LIN {X 0,Y 353.225,Z 325.982,A -85,B 0,C 180,E1 -13406.578,E2 -13406.578} C_VEL
LIN {X 0,Y 353.193,Z 327.589,A -85,B 0,C 180,E1 -13408.86,E2 -13408.86} C_VEL
LIN {X 0,Y 353.218,Z 327.806,A -85,B 0,C 180,E1 -13410,E2 -13410} C_VEL
LIN {X 0,Y 353.193,Z 327.588,A -85,B 0,C 180,E1 -13411.14,E2 -13411.14} C_VEL
LIN {X 0,Y 353.225,Z 325.981,A -85,B 0,C 180,E1 -13413.422,E2 -13413.422} C_VEL
LIN {X 0,Y 353.299,Z 324.582,A -85,B 0,C 180,E1 -13414.564,E2 -13414.564} C_VEL
LIN {X 0,Y 353.388,Z 322.015,A -85,B 0,C 180,E1 -13416.079,E2 -13416.079} C_VEL
LIN {X 0,Y 353.694,Z 317.659,A -85,B 0,C 180,E1 -13417.995,E2 -13417.995} C_VEL
LIN {X 0,Y 354.272,Z 311.542,A -85,B 0,C 180,E1 -13419.996,E2 -13419.996} C_VEL
LIN {X 0,Y 354.955,Z 304.859,A -85,B 0,C 180,E1 -13421.709,E2 -13421.709} C_VEL
LIN {X 0,Y 355.96,Z 296.573,A -85,B 0,C 180,E1 -13423.414,E2 -13423.414} C_VEL
LIN {X 0,Y 356.926,Z 288.08,A -85,B 0,C 180,E1 -13424.831,E2 -13424.831} C_VEL
LIN {X 0,Y 357.965,Z 277.583,A -85,B 0,C 180,E1 -13426.246,E2 -13426.246} C_VEL
LIN {X 0,Y 359.229,Z 265.776,A -85,B 0,C 180,E1 -13427.505,E2 -13427.505} C_VEL
LIN {X 0,Y 359.965,Z 256.498,A -85,B 0,C 180,E1 -13428.294,E2 -13428.294} C_VEL
LIN {X 0,Y 358.531,Z 244.559,A -85,B 0,C 180,E1 -13429.213,E2 -13429.213} C_VEL
LIN {X 0,Y 356.413,Z 231.564,A -85,B 0,C 180,E1 -13429.992,E2 -13429.992} C_VEL
LIN {X 0,Y 354.223,Z 221.02,A -85,B 0,C 180,E1 -13430.496,E2 -13430.496} C_VEL
LIN {X 0,Y 354.747,Z 213.839,A -85,B 0,C 180,E1 -13434.584,E2 -13434.584} C_VEL
LIN {X 0,Y 355.283,Z 207.313,A -85,B 0,C 180,E1 -13438.343,E2 -13438.343} C_VEL
LIN {X 0,Y 355.9,Z 201.27,A -85,B 0,C 180,E1 -13441.883,E2 -13441.883} C_VEL
LIN {X 0,Y 356.363,Z 196.323,A -85,B 0,C 180,E1 -13444.884,E2 -13444.884} C_VEL
LIN {X 0,Y 356.215,Z 191.647,A -85,B 0,C 180,E1 -13447.89,E2 -13447.89} C_VEL
LIN {X 0,Y 355.436,Z 186.73,A -85,B 0,C 180,E1 -13451.291,E2 -13451.291} C_VEL
LIN {X 0,Y 354.794,Z 183.295,A -85,B 0,C 180,E1 -13453.892,E2 -13453.892} C_VEL
LIN {X 0,Y 354.793,Z 183.288,A -85,B 0,C 180,E1 -13457.662,E2 -13457.662} C_VEL
LIN {X 0,Y 354.783,Z 183.293,A -85,B 0,C 180,E1 -13460.662,E2 -13460.662} C_VEL
LIN {X 0,Y 354.819,Z 183.29,A -85,B 0,C 180,E1 -13464.301,E2 -13464.301} C_VEL
LIN {X 0,Y 354.785,Z 183.29,A -85,B 0,C 180,E1 -13467.666,E2 -13467.666} C_VEL
LIN {X 0,Y 354.844,Z 183.283,A -85,B 0,C 180,E1 -13471.618,E2 -13471.618} C_VEL
LIN {X 0,Y 354.896,Z 183.278,A -85,B 0,C 180,E1 -13474.172,E2 -13474.172} C_VEL
LIN {X 0,Y 354.813,Z 183.29,A -85,B 0,C 180,E1 -13477.893,E2 -13477.893} C_VEL
LIN {X 0,Y 354.921,Z 183.275,A -85,B 0,C 180,E1 -13481.891,E2 -13481.891} C_VEL
LIN {X 0,Y 354.94,Z 183.27,A -85,B 0,C 180,E1 -13485.981,E2 -13485.981} C_VEL
LIN {X 0,Y 354.953,Z 183.269,A -85,B 0,C 180,E1 -13489.735,E2 -13489.735} C_VEL
LIN {X 0,Y 355.086,Z 183.257,A -85,B 0,C 180,E1 -13493.18,E2 -13493.18} C_VEL
LIN {X 0,Y 355.24,Z 183.232,A -85,B 0,C 180,E1 -13497.732,E2 -13497.732} C_VEL
LIN {X 0,Y 355.396,Z 183.212,A -85,B 0,C 180,E1 -13500,E2 -13500} C_VEL
LIN {X 0,Y 355.24,Z 183.233,A -85,B 0,C 180,E1 -13502.268,E2 -13502.268} C_VEL
LIN {X 0,Y 355.086,Z 183.254,A -85,B 0,C 180,E1 -13506.82,E2 -13506.82} C_VEL
LIN {X 0,Y 354.953,Z 183.272,A -85,B 0,C 180,E1 -13510.265,E2 -13510.265} C_VEL
LIN {X 0,Y 354.941,Z 183.272,A -85,B 0,C 180,E1 -13514.019,E2 -13514.019} C_VEL
LIN {X 0,Y 354.921,Z 183.277,A -85,B 0,C 180,E1 -13518.109,E2 -13518.109} C_VEL
LIN {X 0,Y 354.833,Z 183.286,A -85,B 0,C 180,E1 -13522.106,E2 -13522.106} C_VEL
LIN {X 0,Y 354.897,Z 183.28,A -85,B 0,C 180,E1 -13525.828,E2 -13525.828} C_VEL
LIN {X 0,Y 354.844,Z 183.286,A -85,B 0,C 180,E1 -13529.68,E2 -13529.68} C_VEL
LIN {X 0,Y 354.805,Z 183.289,A -85,B 0,C 180,E1 -13533.702,E2 -13533.702} C_VEL
LIN {X 0,Y 354.794,Z 183.287,A -85,B 0,C 180,E1 -13536.46,E2 -13536.46} C_VEL
LIN {X 0,Y 354.797,Z 183.291,A -85,B 0,C 180,E1 -13539.419,E2 -13539.419} C_VEL
LIN {X 0,Y 354.787,Z 183.292,A -85,B 0,C 180,E1 -13542.868,E2 -13542.868} C_VEL
LIN {X 0,Y 354.766,Z 183.291,A -85,B 0,C 180,E1 -13546.104,E2 -13546.104} C_VEL
LIN {X 0,Y 354.787,Z 183.291,A -85,B 0,C 180,E1 -13549.18,E2 -13549.18} C_VEL
LIN {X 0,Y 354.775,Z 183.294,A -85,B 0,C 180,E1 -13552.41,E2 -13552.41} C_VEL
LIN {X 0,Y 354.743,Z 183.778,A -85,B 0,C 180,E1 -13553.534,E2 -13553.534} C_VEL
LIN {X 0,Y 354.739,Z 186.75,A -85,B 0,C 180,E1 -13556.315,E2 -13556.315} C_VEL
LIN {X 0,Y 354.595,Z 189.662,A -85,B 0,C 180,E1 -13558.982,E2 -13558.982} C_VEL
LIN {X 0,Y 354.421,Z 192.61,A -85,B 0,C 180,E1 -13561.582,E2 -13561.582} C_VEL
LIN {X 0,Y 354.152,Z 197.072,A -85,B 0,C 180,E1 -13565.372,E2 -13565.372} C_VEL
LIN {X 0,Y 353.952,Z 201.611,A -85,B 0,C 180,E1 -13569.06,E2 -13569.06} C_VEL
LIN {X 0,Y 353.91,Z 202.256,A -85,B 0,C 180,E1 -13569.571,E2 -13569.571} C_VEL
LIN {X 0,Y 357.481,Z 216.111,A -85,B 0,C 180,E1 -13570.331,E2 -13570.331} C_VEL
LIN {X 0,Y 360.044,Z 228.239,A -85,B 0,C 180,E1 -13571.183,E2 -13571.183} C_VEL
LIN {X 0,Y 360.732,Z 234.472,A -85,B 0,C 180,E1 -13571.674,E2 -13571.674} C_VEL
LIN {X 0,Y 359.707,Z 246.144,A -85,B 0,C 180,E1 -13572.665,E2 -13572.665} C_VEL
LIN {X 0,Y 358.615,Z 257.568,A -85,B 0,C 180,E1 -13573.912,E2 -13573.912} C_VEL
LIN {X 0,Y 357.676,Z 267.028,A -85,B 0,C 180,E1 -13575.201,E2 -13575.201} C_VEL
LIN {X 0,Y 356.626,Z 275.52,A -85,B 0,C 180,E1 -13576.612,E2 -13576.612} C_VEL
LIN {X 0,Y 355.618,Z 283.77,A -85,B 0,C 180,E1 -13578.313,E2 -13578.313} C_VEL
LIN {X 0,Y 354.822,Z 290.413,A -85,B 0,C 180,E1 -13580.02,E2 -13580.02} C_VEL
LIN {X 0,Y 354.101,Z 296.5,A -85,B 0,C 180,E1 -13582.014,E2 -13582.014} C_VEL
LIN {X 0,Y 353.768,Z 300.418,A -85,B 0,C 180,E1 -13583.712,E2 -13583.712} C_VEL
LIN {X 0,Y 353.513,Z 303.365,A -85,B 0,C 180,E1 -13585.439,E2 -13585.439} C_VEL
LIN {X 0,Y 353.362,Z 304.764,A -85,B 0,C 180,E1 -13586.58,E2 -13586.58} C_VEL
LIN {X 0,Y 353.273,Z 306.368,A -85,B 0,C 180,E1 -13588.86,E2 -13588.86} C_VEL
LIN {X 0,Y 353.267,Z 306.6,A -85,B 0,C 180,E1 -13590,E2 -13590} C_VEL
LIN {X 0,Y 353.273,Z 306.41,A -85,B 0,C 180,E1 -13591.14,E2 -13591.14} C_VEL
LIN {X 0,Y 353.36,Z 304.86,A -85,B 0,C 180,E1 -13593.421,E2 -13593.421} C_VEL
LIN {X 0,Y 353.51,Z 303.503,A -85,B 0,C 180,E1 -13594.561,E2 -13594.561} C_VEL
LIN {X 0,Y 353.761,Z 300.627,A -85,B 0,C 180,E1 -13596.279,E2 -13596.279} C_VEL
LIN {X 0,Y 354.1,Z 296.754,A -85,B 0,C 180,E1 -13597.986,E2 -13597.986} C_VEL
LIN {X 0,Y 354.647,Z 291.741,A -85,B 0,C 180,E1 -13599.698,E2 -13599.698} C_VEL
LIN {X 0,Y 355.409,Z 285.427,A -85,B 0,C 180,E1 -13601.405,E2 -13601.405} C_VEL
LIN {X 0,Y 356.376,Z 277.523,A -85,B 0,C 180,E1 -13603.108,E2 -13603.108} C_VEL
LIN {X 0,Y 357.603,Z 267.687,A -85,B 0,C 180,E1 -13604.803,E2 -13604.803} C_VEL
LIN {X 0,Y 358.547,Z 258.472,A -85,B 0,C 180,E1 -13606.082,E2 -13606.082} C_VEL
LIN {X 0,Y 359.603,Z 247.14,A -85,B 0,C 180,E1 -13607.34,E2 -13607.34} C_VEL
LIN {X 0,Y 360.72,Z 235.494,A -85,B 0,C 180,E1 -13608.348,E2 -13608.348} C_VEL
LIN {X 0,Y 360.647,Z 231.862,A -85,B 0,C 180,E1 -13608.629,E2 -13608.629} C_VEL
LIN {X 0,Y 358.355,Z 219.915,A -85,B 0,C 180,E1 -13609.528,E2 -13609.528} C_VEL
LIN {X 0,Y 355.219,Z 207.27,A -85,B 0,C 180,E1 -13610.286,E2 -13610.286} C_VEL
LIN {X 0,Y 353.929,Z 202.231,A -85,B 0,C 180,E1 -13610.554,E2 -13610.554} C_VEL
LIN {X 0,Y 354.123,Z 197.861,A -85,B 0,C 180,E1 -13614.087,E2 -13614.087} C_VEL
LIN {X 0,Y 354.324,Z 194.238,A -85,B 0,C 180,E1 -13617.143,E2 -13617.143} C_VEL
LIN {X 0,Y 354.524,Z 191.254,A -85,B 0,C 180,E1 -13619.709,E2 -13619.709} C_VEL
LIN {X 0,Y 354.692,Z 187.612,A -85,B 0,C 180,E1 -13622.983,E2 -13622.983} C_VEL
LIN {X 0,Y 354.809,Z 184.697,A -85,B 0,C 180,E1 -13625.696,E2 -13625.696} C_VEL
LIN {X 0,Y 354.761,Z 183.9,A -85,B 0,C 180,E1 -13626.464,E2 -13626.464} C_VEL
LIN {X 0,Y 354.774,Z 183.292,A -85,B 0,C 180,E1 -13627.851,E2 -13627.851} C_VEL
LIN {X 0,Y 354.122,Z 183.374,A -85,B 0,C 180,E1 -13628.798,E2 -13628.798} C_VEL
LIN {X 0,Y 351.251,Z 183.729,A -85,B 0,C 180,E1 -13630.337,E2 -13630.337} C_VEL
LIN {X 0,Y 348.816,Z 184.035,A -85,B 0,C 180,E1 -13631.583,E2 -13631.583} C_VEL
LIN {X 0,Y 347.784,Z 184.161,A -85,B 0,C 180,E1 -13632.547,E2 -13632.547} C_VEL
LIN {X 0,Y 347.707,Z 184.171,A -85,B 0,C 180,E1 -13632.874,E2 -13632.874} C_VEL
LIN {X 0,Y 347.727,Z 184.17,A -85,B 0,C 180,E1 -13636.686,E2 -13636.686} C_VEL
LIN {X 0,Y 347.73,Z 184.168,A -85,B 0,C 180,E1 -13640.177,E2 -13640.177} C_VEL
LIN {X 0,Y 347.758,Z 184.169,A -85,B 0,C 180,E1 -13642.678,E2 -13642.678} C_VEL
LIN {X 0,Y 347.749,Z 184.165,A -85,B 0,C 180,E1 -13645.956,E2 -13645.956} C_VEL
LIN {X 0,Y 347.75,Z 184.165,A -85,B 0,C 180,E1 -13649.652,E2 -13649.652} C_VEL
LIN {X 0,Y 347.832,Z 184.155,A -85,B 0,C 180,E1 -13653.608,E2 -13653.608} C_VEL
LIN {X 0,Y 347.79,Z 184.165,A -85,B 0,C 180,E1 -13656.162,E2 -13656.162} C_VEL
LIN {X 0,Y 347.816,Z 184.161,A -85,B 0,C 180,E1 -13659.909,E2 -13659.909} C_VEL
LIN {X 0,Y 347.868,Z 184.152,A -85,B 0,C 180,E1 -13662.359,E2 -13662.359} C_VEL
LIN {X 0,Y 347.899,Z 184.15,A -85,B 0,C 180,E1 -13665.971,E2 -13665.971} C_VEL
LIN {X 0,Y 347.897,Z 184.151,A -85,B 0,C 180,E1 -13669.525,E2 -13669.525} C_VEL
LIN {X 0,Y 348.056,Z 184.128,A -85,B 0,C 180,E1 -13673.041,E2 -13673.041} C_VEL
LIN {X 0,Y 348.205,Z 184.11,A -85,B 0,C 180,E1 -13677.686,E2 -13677.686} C_VEL
LIN {X 0,Y 348.348,Z 184.09,A -85,B 0,C 180,E1 -13680,E2 -13680} C_VEL
LIN {X 0,Y 348.205,Z 184.108,A -85,B 0,C 180,E1 -13682.313,E2 -13682.313} C_VEL
LIN {X 0,Y 348.056,Z 184.132,A -85,B 0,C 180,E1 -13686.959,E2 -13686.959} C_VEL
LIN {X 0,Y 347.93,Z 184.146,A -85,B 0,C 180,E1 -13690.474,E2 -13690.474} C_VEL
LIN {X 0,Y 347.9,Z 184.148,A -85,B 0,C 180,E1 -13694.15,E2 -13694.15} C_VEL
LIN {X 0,Y 347.892,Z 184.152,A -85,B 0,C 180,E1 -13698.29,E2 -13698.29} C_VEL
LIN {X 0,Y 347.768,Z 184.163,A -85,B 0,C 180,E1 -13701.626,E2 -13701.626} C_VEL
LIN {X 0,Y 347.812,Z 184.157,A -85,B 0,C 180,E1 -13705.108,E2 -13705.108} C_VEL
LIN {X 0,Y 347.809,Z 184.16,A -85,B 0,C 180,E1 -13707.694,E2 -13707.694} C_VEL
LIN {X 0,Y 347.75,Z 184.167,A -85,B 0,C 180,E1 -13710.348,E2 -13710.348} C_VEL
LIN {X 0,Y 347.749,Z 184.168,A -85,B 0,C 180,E1 -13714.044,E2 -13714.044} C_VEL
LIN {X 0,Y 347.757,Z 184.168,A -85,B 0,C 180,E1 -13717.322,E2 -13717.322} C_VEL
LIN {X 0,Y 347.722,Z 184.169,A -85,B 0,C 180,E1 -13720.299,E2 -13720.299} C_VEL
LIN {X 0,Y 347.724,Z 184.173,A -85,B 0,C 180,E1 -13723.408,E2 -13723.408} C_VEL
LIN {X 0,Y 347.75,Z 184.225,A -85,B 0,C 180,E1 -13725.835,E2 -13725.835} C_VEL
LIN {X 0,Y 348.549,Z 188.551,A -85,B 0,C 180,E1 -13729.07,E2 -13729.07} C_VEL
LIN {X 0,Y 349.139,Z 192.315,A -85,B 0,C 180,E1 -13731.726,E2 -13731.726} C_VEL
LIN {X 0,Y 349.347,Z 196.196,A -85,B 0,C 180,E1 -13734.309,E2 -13734.309} C_VEL
LIN {X 0,Y 349.065,Z 200.582,A -85,B 0,C 180,E1 -13737.07,E2 -13737.07} C_VEL
LIN {X 0,Y 348.487,Z 205.646,A -85,B 0,C 180,E1 -13740.134,E2 -13740.134} C_VEL
LIN {X 0,Y 347.915,Z 211.485,A -85,B 0,C 180,E1 -13743.614,E2 -13743.614} C_VEL
LIN {X 0,Y 347.384,Z 217.947,A -85,B 0,C 180,E1 -13747.394,E2 -13747.394} C_VEL
LIN {X 0,Y 347.232,Z 220.961,A -85,B 0,C 180,E1 -13749.081,E2 -13749.081} C_VEL
LIN {X 0,Y 349.972,Z 234.255,A -85,B 0,C 180,E1 -13749.742,E2 -13749.742} C_VEL
LIN {X 0,Y 351.869,Z 246.195,A -85,B 0,C 180,E1 -13750.522,E2 -13750.522} C_VEL
LIN {X 0,Y 353.131,Z 257.458,A -85,B 0,C 180,E1 -13751.432,E2 -13751.432} C_VEL
LIN {X 0,Y 352.183,Z 268.48,A -85,B 0,C 180,E1 -13752.432,E2 -13752.432} C_VEL
LIN {X 0,Y 350.898,Z 279.731,A -85,B 0,C 180,E1 -13753.716,E2 -13753.716} C_VEL
LIN {X 0,Y 349.791,Z 289.701,A -85,B 0,C 180,E1 -13755.157,E2 -13755.157} C_VEL
LIN {X 0,Y 348.66,Z 299.37,A -85,B 0,C 180,E1 -13756.893,E2 -13756.893} C_VEL
LIN {X 0,Y 347.698,Z 307.067,A -85,B 0,C 180,E1 -13758.634,E2 -13758.634} C_VEL
LIN {X 0,Y 346.954,Z 314.168,A -85,B 0,C 180,E1 -13760.674,E2 -13760.674} C_VEL
LIN {X 0,Y 346.505,Z 318.893,A -85,B 0,C 180,E1 -13762.424,E2 -13762.424} C_VEL
LIN {X 0,Y 346.25,Z 322.506,A -85,B 0,C 180,E1 -13764.175,E2 -13764.175} C_VEL
LIN {X 0,Y 346.215,Z 324.372,A -85,B 0,C 180,E1 -13765.342,E2 -13765.342} C_VEL
LIN {X 0,Y 346.15,Z 325.77,A -85,B 0,C 180,E1 -13766.508,E2 -13766.508} C_VEL
LIN {X 0,Y 346.094,Z 327.376,A -85,B 0,C 180,E1 -13768.836,E2 -13768.836} C_VEL
LIN {X 0,Y 346.121,Z 327.593,A -85,B 0,C 180,E1 -13770,E2 -13770} C_VEL
LIN {X 0,Y 346.094,Z 327.375,A -85,B 0,C 180,E1 -13771.163,E2 -13771.163} C_VEL
LIN {X 0,Y 346.15,Z 325.767,A -85,B 0,C 180,E1 -13773.492,E2 -13773.492} C_VEL
LIN {X 0,Y 346.216,Z 324.368,A -85,B 0,C 180,E1 -13774.657,E2 -13774.657} C_VEL
LIN {X 0,Y 346.279,Z 322.148,A -85,B 0,C 180,E1 -13776.015,E2 -13776.015} C_VEL
LIN {X 0,Y 346.646,Z 317.444,A -85,B 0,C 180,E1 -13778.159,E2 -13778.159} C_VEL
LIN {X 0,Y 347.257,Z 311.326,A -85,B 0,C 180,E1 -13780.2,E2 -13780.2} C_VEL
LIN {X 0,Y 347.985,Z 304.643,A -85,B 0,C 180,E1 -13781.947,E2 -13781.947} C_VEL
LIN {X 0,Y 349.033,Z 296.357,A -85,B 0,C 180,E1 -13783.685,E2 -13783.685} C_VEL
LIN {X 0,Y 350.04,Z 287.863,A -85,B 0,C 180,E1 -13785.13,E2 -13785.13} C_VEL
LIN {X 0,Y 351.12,Z 277.366,A -85,B 0,C 180,E1 -13786.572,E2 -13786.572} C_VEL
LIN {X 0,Y 352.437,Z 265.558,A -85,B 0,C 180,E1 -13787.854,E2 -13787.854} C_VEL
LIN {X 0,Y 353.105,Z 257.375,A -85,B 0,C 180,E1 -13788.569,E2 -13788.569} C_VEL
LIN {X 0,Y 351.776,Z 245.669,A -85,B 0,C 180,E1 -13789.51,E2 -13789.51} C_VEL
LIN {X 0,Y 349.662,Z 232.674,A -85,B 0,C 180,E1 -13790.339,E2 -13790.339} C_VEL
LIN {X 0,Y 347.208,Z 220.824,A -85,B 0,C 180,E1 -13790.92,E2 -13790.92} C_VEL
LIN {X 0,Y 347.669,Z 214.624,A -85,B 0,C 180,E1 -13794.541,E2 -13794.541} C_VEL
LIN {X 0,Y 348.243,Z 208.221,A -85,B 0,C 180,E1 -13798.311,E2 -13798.311} C_VEL
LIN {X 0,Y 348.92,Z 201.708,A -85,B 0,C 180,E1 -13802.224,E2 -13802.224} C_VEL
LIN {X 0,Y 349.36,Z 197.247,A -85,B 0,C 180,E1 -13804.984,E2 -13804.984} C_VEL
LIN {X 0,Y 349.307,Z 193.958,A -85,B 0,C 180,E1 -13807.127,E2 -13807.127} C_VEL
LIN {X 0,Y 348.725,Z 189.58,A -85,B 0,C 180,E1 -13810.158,E2 -13810.158} C_VEL
LIN {X 0,Y 347.948,Z 185.227,A -85,B 0,C 180,E1 -13813.372,E2 -13813.372} C_VEL
LIN {X 0,Y 347.734,Z 184.173,A -85,B 0,C 180,E1 -13814.306,E2 -13814.306} C_VEL
LIN {X 0,Y 347.748,Z 184.171,A -85,B 0,C 180,E1 -13818.397,E2 -13818.397} C_VEL
LIN {X 0,Y 347.762,Z 184.166,A -85,B 0,C 180,E1 -13822.013,E2 -13822.013} C_VEL
LIN {X 0,Y 347.742,Z 184.166,A -85,B 0,C 180,E1 -13825.536,E2 -13825.536} C_VEL
LIN {X 0,Y 347.743,Z 184.171,A -85,B 0,C 180,E1 -13828.3,E2 -13828.3} C_VEL
LIN {X 0,Y 347.777,Z 184.162,A -85,B 0,C 180,E1 -13830.987,E2 -13830.987} C_VEL
LIN {X 0,Y 347.829,Z 184.158,A -85,B 0,C 180,E1 -13833.607,E2 -13833.607} C_VEL
LIN {X 0,Y 347.783,Z 184.164,A -85,B 0,C 180,E1 -13836.161,E2 -13836.161} C_VEL
LIN {X 0,Y 347.809,Z 184.161,A -85,B 0,C 180,E1 -13839.909,E2 -13839.909} C_VEL
LIN {X 0,Y 347.864,Z 184.151,A -85,B 0,C 180,E1 -13842.359,E2 -13842.359} C_VEL
LIN {X 0,Y 347.895,Z 184.148,A -85,B 0,C 180,E1 -13845.971,E2 -13845.971} C_VEL
LIN {X 0,Y 347.893,Z 184.15,A -85,B 0,C 180,E1 -13849.525,E2 -13849.525} C_VEL
LIN {X 0,Y 348.053,Z 184.132,A -85,B 0,C 180,E1 -13853.041,E2 -13853.041} C_VEL
LIN {X 0,Y 348.202,Z 184.109,A -85,B 0,C 180,E1 -13857.687,E2 -13857.687} C_VEL
LIN {X 0,Y 348.344,Z 184.091,A -85,B 0,C 180,E1 -13860,E2 -13860} C_VEL
LIN {X 0,Y 348.202,Z 184.11,A -85,B 0,C 180,E1 -13862.314,E2 -13862.314} C_VEL
LIN {X 0,Y 348.052,Z 184.129,A -85,B 0,C 180,E1 -13866.959,E2 -13866.959} C_VEL
LIN {X 0,Y 347.893,Z 184.152,A -85,B 0,C 180,E1 -13870.476,E2 -13870.476} C_VEL
LIN {X 0,Y 347.896,Z 184.151,A -85,B 0,C 180,E1 -13874.15,E2 -13874.15} C_VEL
LIN {X 0,Y 347.89,Z 184.151,A -85,B 0,C 180,E1 -13878.291,E2 -13878.291} C_VEL
LIN {X 0,Y 347.787,Z 184.163,A -85,B 0,C 180,E1 -13881.635,E2 -13881.635} C_VEL
LIN {X 0,Y 347.81,Z 184.158,A -85,B 0,C 180,E1 -13885.109,E2 -13885.109} C_VEL
LIN {X 0,Y 347.806,Z 184.163,A -85,B 0,C 180,E1 -13887.694,E2 -13887.694} C_VEL
LIN {X 0,Y 347.759,Z 184.164,A -85,B 0,C 180,E1 -13890.347,E2 -13890.347} C_VEL
LIN {X 0,Y 347.743,Z 184.166,A -85,B 0,C 180,E1 -13894.464,E2 -13894.464} C_VEL
LIN {X 0,Y 347.762,Z 184.164,A -85,B 0,C 180,E1 -13897.987,E2 -13897.987} C_VEL
LIN {X 0,Y 347.749,Z 184.165,A -85,B 0,C 180,E1 -13901.831,E2 -13901.831} C_VEL
LIN {X 0,Y 347.705,Z 184.176,A -85,B 0,C 180,E1 -13905.027,E2 -13905.027} C_VEL
LIN {X 0,Y 347.75,Z 184.167,A -85,B 0,C 180,E1 -13908.398,E2 -13908.398} C_VEL
LIN {X 0,Y 347.755,Z 184.166,A -85,B 0,C 180,E1 -13912.016,E2 -13912.016} C_VEL
LIN {X 0,Y 347.697,Z 184.178,A -85,B 0,C 180,E1 -13912.672,E2 -13912.672} C_VEL
LIN {X 0,Y 347.743,Z 185.405,A -85,B 0,C 180,E1 -13914.12,E2 -13914.12} C_VEL
LIN {X 0,Y 347.649,Z 188.379,A -85,B 0,C 180,E1 -13916.919,E2 -13916.919} C_VEL
LIN {X 0,Y 347.475,Z 192.197,A -85,B 0,C 180,E1 -13920.426,E2 -13920.426} C_VEL
LIN {X 0,Y 347.226,Z 195.774,A -85,B 0,C 180,E1 -13923.559,E2 -13923.559} C_VEL
LIN {X 0,Y 347.102,Z 198.77,A -85,B 0,C 180,E1 -13926.112,E2 -13926.112} C_VEL
LIN {X 0,Y 346.899,Z 202.462,A -85,B 0,C 180,E1 -13929.134,E2 -13929.134} C_VEL
LIN {X 0,Y 350.567,Z 216.542,A -85,B 0,C 180,E1 -13929.937,E2 -13929.937} C_VEL
LIN {X 0,Y 353.199,Z 229.136,A -85,B 0,C 180,E1 -13930.85,E2 -13930.85} C_VEL
LIN {X 0,Y 353.996,Z 234.818,A -85,B 0,C 180,E1 -13931.322,E2 -13931.322} C_VEL
LIN {X 0,Y 352.93,Z 246.363,A -85,B 0,C 180,E1 -13932.322,E2 -13932.322} C_VEL
LIN {X 0,Y 351.76,Z 258.047,A -85,B 0,C 180,E1 -13933.623,E2 -13933.623} C_VEL
LIN {X 0,Y 350.823,Z 267.245,A -85,B 0,C 180,E1 -13934.905,E2 -13934.905} C_VEL
LIN {X 0,Y 349.732,Z 275.736,A -85,B 0,C 180,E1 -13936.343,E2 -13936.343} C_VEL
LIN {X 0,Y 348.67,Z 283.985,A -85,B 0,C 180,E1 -13938.077,E2 -13938.077} C_VEL
LIN {X 0,Y 347.818,Z 290.629,A -85,B 0,C 180,E1 -13939.817,E2 -13939.817} C_VEL
LIN {X 0,Y 347.078,Z 296.714,A -85,B 0,C 180,E1 -13941.852,E2 -13941.852} C_VEL
LIN {X 0,Y 346.8,Z 299.866,A -85,B 0,C 180,E1 -13943.218,E2 -13943.218} C_VEL
LIN {X 0,Y 346.454,Z 303.579,A -85,B 0,C 180,E1 -13945.346,E2 -13945.346} C_VEL
LIN {X 0,Y 346.285,Z 304.977,A -85,B 0,C 180,E1 -13946.51,E2 -13946.51} C_VEL
LIN {X 0,Y 346.176,Z 306.582,A -85,B 0,C 180,E1 -13948.837,E2 -13948.837} C_VEL
LIN {X 0,Y 346.171,Z 306.813,A -85,B 0,C 180,E1 -13950,E2 -13950} C_VEL
LIN {X 0,Y 346.176,Z 306.623,A -85,B 0,C 180,E1 -13951.164,E2 -13951.164} C_VEL
LIN {X 0,Y 346.284,Z 305.072,A -85,B 0,C 180,E1 -13953.491,E2 -13953.491} C_VEL
LIN {X 0,Y 346.451,Z 303.715,A -85,B 0,C 180,E1 -13954.655,E2 -13954.655} C_VEL
LIN {X 0,Y 346.798,Z 300.089,A -85,B 0,C 180,E1 -13956.779,E2 -13956.779} C_VEL
LIN {X 0,Y 347.244,Z 295.409,A -85,B 0,C 180,E1 -13958.731,E2 -13958.731} C_VEL
LIN {X 0,Y 348.037,Z 288.974,A -85,B 0,C 180,E1 -13960.766,E2 -13960.766} C_VEL
LIN {X 0,Y 348.965,Z 281.9,A -85,B 0,C 180,E1 -13962.504,E2 -13962.504} C_VEL
LIN {X 0,Y 350.097,Z 273.085,A -85,B 0,C 180,E1 -13964.236,E2 -13964.236} C_VEL
LIN {X 0,Y 351.219,Z 264.15,A -85,B 0,C 180,E1 -13965.655,E2 -13965.655} C_VEL
LIN {X 0,Y 352.179,Z 254.399,A -85,B 0,C 180,E1 -13966.924,E2 -13966.924} C_VEL
LIN {X 0,Y 353.195,Z 244.446,A -85,B 0,C 180,E1 -13967.965,E2 -13967.965} C_VEL
LIN {X 0,Y 353.965,Z 233.582,A -85,B 0,C 180,E1 -13968.879,E2 -13968.879} C_VEL
LIN {X 0,Y 351.613,Z 221.039,A -85,B 0,C 180,E1 -13969.865,E2 -13969.865} C_VEL
LIN {X 0,Y 348.482,Z 208.389,A -85,B 0,C 180,E1 -13970.664,E2 -13970.664} C_VEL
LIN {X 0,Y 346.897,Z 202.432,A -85,B 0,C 180,E1 -13970.999,E2 -13970.999} C_VEL
LIN {X 0,Y 347.07,Z 198.393,A -85,B 0,C 180,E1 -13974.324,E2 -13974.324} C_VEL
LIN {X 0,Y 347.315,Z 194.433,A -85,B 0,C 180,E1 -13977.737,E2 -13977.737} C_VEL
LIN {X 0,Y 347.507,Z 191.435,A -85,B 0,C 180,E1 -13980.371,E2 -13980.371} C_VEL
LIN {X 0,Y 347.738,Z 187.462,A -85,B 0,C 180,E1 -13984.041,E2 -13984.041} C_VEL
LIN {X 0,Y 347.774,Z 185.343,A -85,B 0,C 180,E1 -13986.065,E2 -13986.065} C_VEL
LIN {X 0,Y 347.697,Z 184.177,A -85,B 0,C 180,E1 -13987.329,E2 -13987.329} C_VEL
LIN {X 0,Y 347.698,Z 184.171,A -85,B 0,C 180,E1 -13990.302,E2 -13990.302} C_VEL
LIN {X 0,Y 347.707,Z 184.171,A -85,B 0,C 180,E1 -13992.874,E2 -13992.874} C_VEL
LIN {X 0,Y 347.07,Z 184.254,A -85,B 0,C 180,E1 -13993.841,E2 -13993.841} C_VEL
LIN {X 0,Y 344.259,Z 184.605,A -85,B 0,C 180,E1 -13995.415,E2 -13995.415} C_VEL
LIN {X 0,Y 341.85,Z 184.902,A -85,B 0,C 180,E1 -13996.689,E2 -13996.689} C_VEL
LIN {X 0,Y 340.794,Z 185.033,A -85,B 0,C 180,E1 -13997.674,E2 -13997.674} C_VEL
LIN {X 0,Y 340.697,Z 185.044,A -85,B 0,C 180,E1 -13998.008,E2 -13998.008} C_VEL
LIN {X 0,Y 340.721,Z 185.041,A -85,B 0,C 180,E1 -14001.771,E2 -14001.771} C_VEL
LIN {X 0,Y 340.724,Z 185.04,A -85,B 0,C 180,E1 -14005.595,E2 -14005.595} C_VEL
LIN {X 0,Y 340.699,Z 185.045,A -85,B 0,C 180,E1 -14008.955,E2 -14008.955} C_VEL
LIN {X 0,Y 340.805,Z 185.03,A -85,B 0,C 180,E1 -14013.02,E2 -14013.02} C_VEL
LIN {X 0,Y 340.757,Z 185.037,A -85,B 0,C 180,E1 -14015.638,E2 -14015.638} C_VEL
LIN {X 0,Y 340.747,Z 185.038,A -85,B 0,C 180,E1 -14019.474,E2 -14019.474} C_VEL
LIN {X 0,Y 340.859,Z 185.028,A -85,B 0,C 180,E1 -14021.984,E2 -14021.984} C_VEL
LIN {X 0,Y 340.871,Z 185.027,A -85,B 0,C 180,E1 -14025.705,E2 -14025.705} C_VEL
LIN {X 0,Y 340.849,Z 185.027,A -85,B 0,C 180,E1 -14029.305,E2 -14029.305} C_VEL
LIN {X 0,Y 341.003,Z 185.006,A -85,B 0,C 180,E1 -14032.897,E2 -14032.897} C_VEL
LIN {X 0,Y 341.166,Z 184.987,A -85,B 0,C 180,E1 -14037.639,E2 -14037.639} C_VEL
LIN {X 0,Y 341.298,Z 184.969,A -85,B 0,C 180,E1 -14040,E2 -14040} C_VEL
LIN {X 0,Y 341.167,Z 184.985,A -85,B 0,C 180,E1 -14042.361,E2 -14042.361} C_VEL
LIN {X 0,Y 341.003,Z 185.009,A -85,B 0,C 180,E1 -14047.103,E2 -14047.103} C_VEL
LIN {X 0,Y 340.873,Z 185.027,A -85,B 0,C 180,E1 -14050.694,E2 -14050.694} C_VEL
LIN {X 0,Y 340.864,Z 185.026,A -85,B 0,C 180,E1 -14054.325,E2 -14054.325} C_VEL
LIN {X 0,Y 340.838,Z 185.031,A -85,B 0,C 180,E1 -14058.466,E2 -14058.466} C_VEL
LIN {X 0,Y 340.719,Z 185.043,A -85,B 0,C 180,E1 -14061.842,E2 -14061.842} C_VEL
LIN {X 0,Y 340.773,Z 185.036,A -85,B 0,C 180,E1 -14065.664,E2 -14065.664} C_VEL
LIN {X 0,Y 340.729,Z 185.042,A -85,B 0,C 180,E1 -14068.321,E2 -14068.321} C_VEL
LIN {X 0,Y 340.699,Z 185.044,A -85,B 0,C 180,E1 -14071.045,E2 -14071.045} C_VEL
LIN {X 0,Y 340.718,Z 185.044,A -85,B 0,C 180,E1 -14075.279,E2 -14075.279} C_VEL
LIN {X 0,Y 340.694,Z 185.045,A -85,B 0,C 180,E1 -14078.383,E2 -14078.383} C_VEL
LIN {X 0,Y 340.7,Z 185.046,A -85,B 0,C 180,E1 -14082.045,E2 -14082.045} C_VEL
LIN {X 0,Y 340.714,Z 185.118,A -85,B 0,C 180,E1 -14085.466,E2 -14085.466} C_VEL
LIN {X 0,Y 341.497,Z 189.479,A -85,B 0,C 180,E1 -14088.81,E2 -14088.81} C_VEL
LIN {X 0,Y 342.161,Z 193.851,A -85,B 0,C 180,E1 -14091.961,E2 -14091.961} C_VEL
LIN {X 0,Y 342.332,Z 198.232,A -85,B 0,C 180,E1 -14094.912,E2 -14094.912} C_VEL
LIN {X 0,Y 341.784,Z 203.704,A -85,B 0,C 180,E1 -14098.375,E2 -14098.375} C_VEL
LIN {X 0,Y 341.06,Z 210.223,A -85,B 0,C 180,E1 -14102.384,E2 -14102.384} C_VEL
LIN {X 0,Y 340.449,Z 216.677,A -85,B 0,C 180,E1 -14106.262,E2 -14106.262} C_VEL
LIN {X 0,Y 340.192,Z 220.823,A -85,B 0,C 180,E1 -14108.629,E2 -14108.629} C_VEL
LIN {X 0,Y 342.938,Z 233.732,A -85,B 0,C 180,E1 -14109.292,E2 -14109.292} C_VEL
LIN {X 0,Y 344.975,Z 246.283,A -85,B 0,C 180,E1 -14110.137,E2 -14110.137} C_VEL
LIN {X 0,Y 346.202,Z 257.243,A -85,B 0,C 180,E1 -14111.046,E2 -14111.046} C_VEL
LIN {X 0,Y 345.911,Z 263.877,A -85,B 0,C 180,E1 -14111.644,E2 -14111.644} C_VEL
LIN {X 0,Y 344.606,Z 274.854,A -85,B 0,C 180,E1 -14112.799,E2 -14112.799} C_VEL
LIN {X 0,Y 343.477,Z 284.578,A -85,B 0,C 180,E1 -14114.088,E2 -14114.088} C_VEL
LIN {X 0,Y 342.308,Z 294.591,A -85,B 0,C 180,E1 -14115.737,E2 -14115.737} C_VEL
LIN {X 0,Y 341.147,Z 303.218,A -85,B 0,C 180,E1 -14117.507,E2 -14117.507} C_VEL
LIN {X 0,Y 340.36,Z 310.12,A -85,B 0,C 180,E1 -14119.29,E2 -14119.29} C_VEL
LIN {X 0,Y 339.742,Z 315.652,A -85,B 0,C 180,E1 -14121.074,E2 -14121.074} C_VEL
LIN {X 0,Y 339.352,Z 319.994,A -85,B 0,C 180,E1 -14122.862,E2 -14122.862} C_VEL
LIN {X 0,Y 339.17,Z 322.293,A -85,B 0,C 180,E1 -14124.053,E2 -14124.053} C_VEL
LIN {X 0,Y 339.115,Z 324.158,A -85,B 0,C 180,E1 -14125.245,E2 -14125.245} C_VEL
LIN {X 0,Y 339.077,Z 325.557,A -85,B 0,C 180,E1 -14126.435,E2 -14126.435} C_VEL
LIN {X 0,Y 338.998,Z 327.164,A -85,B 0,C 180,E1 -14128.812,E2 -14128.812} C_VEL
LIN {X 0,Y 339.025,Z 327.38,A -85,B 0,C 180,E1 -14130,E2 -14130} C_VEL
LIN {X 0,Y 338.998,Z 327.162,A -85,B 0,C 180,E1 -14131.188,E2 -14131.188} C_VEL
LIN {X 0,Y 339.077,Z 325.554,A -85,B 0,C 180,E1 -14133.565,E2 -14133.565} C_VEL
LIN {X 0,Y 339.115,Z 324.153,A -85,B 0,C 180,E1 -14134.755,E2 -14134.755} C_VEL
LIN {X 0,Y 339.25,Z 321.21,A -85,B 0,C 180,E1 -14136.542,E2 -14136.542} C_VEL
LIN {X 0,Y 339.592,Z 317.229,A -85,B 0,C 180,E1 -14138.329,E2 -14138.329} C_VEL
LIN {X 0,Y 340.233,Z 311.111,A -85,B 0,C 180,E1 -14140.413,E2 -14140.413} C_VEL
LIN {X 0,Y 341.012,Z 304.428,A -85,B 0,C 180,E1 -14142.195,E2 -14142.195} C_VEL
LIN {X 0,Y 342.114,Z 296.141,A -85,B 0,C 180,E1 -14143.968,E2 -14143.968} C_VEL
LIN {X 0,Y 343.276,Z 286.478,A -85,B 0,C 180,E1 -14145.618,E2 -14145.618} C_VEL
LIN {X 0,Y 344.431,Z 275.971,A -85,B 0,C 180,E1 -14147.056,E2 -14147.056} C_VEL
LIN {X 0,Y 345.679,Z 265.34,A -85,B 0,C 180,E1 -14148.215,E2 -14148.215} C_VEL
LIN {X 0,Y 346.283,Z 258.929,A -85,B 0,C 180,E1 -14148.795,E2 -14148.795} C_VEL
LIN {X 0,Y 345.088,Z 247.403,A -85,B 0,C 180,E1 -14149.77,E2 -14149.77} C_VEL
LIN {X 0,Y 343.092,Z 234.647,A -85,B 0,C 180,E1 -14150.642,E2 -14150.642} C_VEL
LIN {X 0,Y 340.343,Z 221.809,A -85,B 0,C 180,E1 -14151.325,E2 -14151.325} C_VEL
LIN {X 0,Y 340.176,Z 220.528,A -85,B 0,C 180,E1 -14151.424,E2 -14151.424} C_VEL
LIN {X 0,Y 340.623,Z 214.91,A -85,B 0,C 180,E1 -14154.791,E2 -14154.791} C_VEL
LIN {X 0,Y 341.188,Z 209.125,A -85,B 0,C 180,E1 -14158.279,E2 -14158.279} C_VEL
LIN {X 0,Y 341.777,Z 203.681,A -85,B 0,C 180,E1 -14161.625,E2 -14161.625} C_VEL
LIN {X 0,Y 342.339,Z 198.193,A -85,B 0,C 180,E1 -14165.087,E2 -14165.087} C_VEL
LIN {X 0,Y 342.157,Z 193.801,A -85,B 0,C 180,E1 -14168.039,E2 -14168.039} C_VEL
LIN {X 0,Y 341.496,Z 189.427,A -85,B 0,C 180,E1 -14171.19,E2 -14171.19} C_VEL
LIN {X 0,Y 340.688,Z 185.052,A -85,B 0,C 180,E1 -14174.635,E2 -14174.635} C_VEL
LIN {X 0,Y 340.681,Z 185.051,A -85,B 0,C 180,E1 -14178.69,E2 -14178.69} C_VEL
LIN {X 0,Y 340.718,Z 185.042,A -85,B 0,C 180,E1 -14181.771,E2 -14181.771} C_VEL
LIN {X 0,Y 340.721,Z 185.041,A -85,B 0,C 180,E1 -14185.595,E2 -14185.595} C_VEL
LIN {X 0,Y 340.696,Z 185.044,A -85,B 0,C 180,E1 -14188.955,E2 -14188.955} C_VEL
LIN {X 0,Y 340.801,Z 185.031,A -85,B 0,C 180,E1 -14193.02,E2 -14193.02} C_VEL
LIN {X 0,Y 340.752,Z 185.04,A -85,B 0,C 180,E1 -14195.638,E2 -14195.638} C_VEL
LIN {X 0,Y 340.735,Z 185.042,A -85,B 0,C 180,E1 -14199.473,E2 -14199.473} C_VEL
LIN {X 0,Y 340.856,Z 185.026,A -85,B 0,C 180,E1 -14201.984,E2 -14201.984} C_VEL
LIN {X 0,Y 340.867,Z 185.026,A -85,B 0,C 180,E1 -14205.705,E2 -14205.705} C_VEL
LIN {X 0,Y 340.845,Z 185.029,A -85,B 0,C 180,E1 -14209.305,E2 -14209.305} C_VEL
LIN {X 0,Y 340.999,Z 185.009,A -85,B 0,C 180,E1 -14212.897,E2 -14212.897} C_VEL
LIN {X 0,Y 341.164,Z 184.986,A -85,B 0,C 180,E1 -14217.639,E2 -14217.639} C_VEL
LIN {X 0,Y 341.295,Z 184.969,A -85,B 0,C 180,E1 -14220,E2 -14220} C_VEL
LIN {X 0,Y 341.164,Z 184.987,A -85,B 0,C 180,E1 -14222.361,E2 -14222.361} C_VEL
LIN {X 0,Y 340.999,Z 185.007,A -85,B 0,C 180,E1 -14227.103,E2 -14227.103} C_VEL
LIN {X 0,Y 340.845,Z 185.028,A -85,B 0,C 180,E1 -14230.695,E2 -14230.695} C_VEL
LIN {X 0,Y 340.861,Z 185.028,A -85,B 0,C 180,E1 -14234.325,E2 -14234.325} C_VEL
LIN {X 0,Y 340.836,Z 185.028,A -85,B 0,C 180,E1 -14238.467,E2 -14238.467} C_VEL
LIN {X 0,Y 340.752,Z 185.041,A -85,B 0,C 180,E1 -14241.857,E2 -14241.857} C_VEL
LIN {X 0,Y 340.77,Z 185.039,A -85,B 0,C 180,E1 -14245.665,E2 -14245.665} C_VEL
LIN {X 0,Y 340.727,Z 185.04,A -85,B 0,C 180,E1 -14248.321,E2 -14248.321} C_VEL
LIN {X 0,Y 340.701,Z 185.044,A -85,B 0,C 180,E1 -14251.045,E2 -14251.045} C_VEL
LIN {X 0,Y 340.716,Z 185.046,A -85,B 0,C 180,E1 -14255.279,E2 -14255.279} C_VEL
LIN {X 0,Y 340.693,Z 185.045,A -85,B 0,C 180,E1 -14258.383,E2 -14258.383} C_VEL
LIN {X 0,Y 340.698,Z 185.044,A -85,B 0,C 180,E1 -14262.046,E2 -14262.046} C_VEL
LIN {X 0,Y 340.651,Z 185.05,A -85,B 0,C 180,E1 -14266.227,E2 -14266.227} C_VEL
LIN {X 0,Y 340.687,Z 185.046,A -85,B 0,C 180,E1 -14269.754,E2 -14269.754} C_VEL
LIN {X 0,Y 340.719,Z 185.042,A -85,B 0,C 180,E1 -14271.771,E2 -14271.771} C_VEL
LIN {X 0,Y 340.687,Z 185.892,A -85,B 0,C 180,E1 -14273.565,E2 -14273.565} C_VEL
LIN {X 0,Y 340.648,Z 188.527,A -85,B 0,C 180,E1 -14276.149,E2 -14276.149} C_VEL
LIN {X 0,Y 340.504,Z 191.498,A -85,B 0,C 180,E1 -14278.936,E2 -14278.936} C_VEL
LIN {X 0,Y 340.265,Z 195.593,A -85,B 0,C 180,E1 -14282.641,E2 -14282.641} C_VEL
LIN {X 0,Y 339.979,Z 200.504,A -85,B 0,C 180,E1 -14286.874,E2 -14286.874} C_VEL
LIN {X 0,Y 339.867,Z 202.676,A -85,B 0,C 180,E1 -14288.68,E2 -14288.68} C_VEL
LIN {X 0,Y 343.572,Z 216.672,A -85,B 0,C 180,E1 -14289.505,E2 -14289.505} C_VEL
LIN {X 0,Y 345.924,Z 227.602,A -85,B 0,C 180,E1 -14290.309,E2 -14290.309} C_VEL
LIN {X 0,Y 347.181,Z 235.182,A -85,B 0,C 180,E1 -14290.953,E2 -14290.953} C_VEL
LIN {X 0,Y 346.179,Z 246.581,A -85,B 0,C 180,E1 -14291.965,E2 -14291.965} C_VEL
LIN {X 0,Y 344.989,Z 257.792,A -85,B 0,C 180,E1 -14293.231,E2 -14293.231} C_VEL
LIN {X 0,Y 343.981,Z 267.461,A -85,B 0,C 180,E1 -14294.597,E2 -14294.597} C_VEL
LIN {X 0,Y 342.831,Z 275.952,A -85,B 0,C 180,E1 -14296.062,E2 -14296.062} C_VEL
LIN {X 0,Y 341.736,Z 284.2,A -85,B 0,C 180,E1 -14297.831,E2 -14297.831} C_VEL
LIN {X 0,Y 340.838,Z 290.844,A -85,B 0,C 180,E1 -14299.606,E2 -14299.606} C_VEL
LIN {X 0,Y 340.041,Z 296.929,A -85,B 0,C 180,E1 -14301.682,E2 -14301.682} C_VEL
LIN {X 0,Y 339.729,Z 300.354,A -85,B 0,C 180,E1 -14303.209,E2 -14303.209} C_VEL
LIN {X 0,Y 339.397,Z 303.792,A -85,B 0,C 180,E1 -14305.249,E2 -14305.249} C_VEL
LIN {X 0,Y 339.212,Z 305.19,A -85,B 0,C 180,E1 -14306.437,E2 -14306.437} C_VEL
LIN {X 0,Y 339.079,Z 306.795,A -85,B 0,C 180,E1 -14308.813,E2 -14308.813} C_VEL
LIN {X 0,Y 339.075,Z 307.026,A -85,B 0,C 180,E1 -14310,E2 -14310} C_VEL
LIN {X 0,Y 339.079,Z 306.836,A -85,B 0,C 180,E1 -14311.188,E2 -14311.188} C_VEL
LIN {X 0,Y 339.211,Z 305.284,A -85,B 0,C 180,E1 -14313.564,E2 -14313.564} C_VEL
LIN {X 0,Y 339.394,Z 303.927,A -85,B 0,C 180,E1 -14314.752,E2 -14314.752} C_VEL
LIN {X 0,Y 339.727,Z 300.575,A -85,B 0,C 180,E1 -14316.788,E2 -14316.788} C_VEL
LIN {X 0,Y 340.222,Z 295.621,A -85,B 0,C 180,E1 -14318.913,E2 -14318.913} C_VEL
LIN {X 0,Y 341.045,Z 289.186,A -85,B 0,C 180,E1 -14320.989,E2 -14320.989} C_VEL
LIN {X 0,Y 342.002,Z 282.112,A -85,B 0,C 180,E1 -14322.763,E2 -14322.763} C_VEL
LIN {X 0,Y 343.221,Z 273.295,A -85,B 0,C 180,E1 -14324.527,E2 -14324.527} C_VEL
LIN {X 0,Y 344.359,Z 264.572,A -85,B 0,C 180,E1 -14325.942,E2 -14325.942} C_VEL
LIN {X 0,Y 345.403,Z 254.607,A -85,B 0,C 180,E1 -14327.267,E2 -14327.267} C_VEL
LIN {X 0,Y 346.472,Z 244.652,A -85,B 0,C 180,E1 -14328.325,E2 -14328.325} C_VEL
LIN {X 0,Y 347.257,Z 235.188,A -85,B 0,C 180,E1 -14329.148,E2 -14329.148} C_VEL
LIN {X 0,Y 345.187,Z 223.765,A -85,B 0,C 180,E1 -14330.099,E2 -14330.099} C_VEL
LIN {X 0,Y 342.045,Z 210.626,A -85,B 0,C 180,E1 -14330.984,E2 -14330.984} C_VEL
LIN {X 0,Y 339.835,Z 202.67,A -85,B 0,C 180,E1 -14331.438,E2 -14331.438} C_VEL
LIN {X 0,Y 340.028,Z 198.926,A -85,B 0,C 180,E1 -14334.573,E2 -14334.573} C_VEL
LIN {X 0,Y 340.324,Z 194.617,A -85,B 0,C 180,E1 -14338.358,E2 -14338.358} C_VEL
LIN {X 0,Y 340.506,Z 191.619,A -85,B 0,C 180,E1 -14341.064,E2 -14341.064} C_VEL
LIN {X 0,Y 340.724,Z 188.091,A -85,B 0,C 180,E1 -14344.404,E2 -14344.404} C_VEL
LIN {X 0,Y 340.679,Z 185.696,A -85,B 0,C 180,E1 -14346.745,E2 -14346.745} C_VEL
LIN {X 0,Y 340.684,Z 185.047,A -85,B 0,C 180,E1 -14348.38,E2 -14348.38} C_VEL
LIN {X 0,Y 340.695,Z 185.044,A -85,B 0,C 180,E1 -14352.044,E2 -14352.044} C_VEL
LIN {X 0,Y 340.653,Z 185.049,A -85,B 0,C 180,E1 -14356.227,E2 -14356.227} C_VEL
LIN {X 0,Y 340.697,Z 185.044,A -85,B 0,C 180,E1 -14358.008,E2 -14358.008} C_VEL
LIN {X 0,Y 340.004,Z 185.135,A -85,B 0,C 180,E1 -14358.995,E2 -14358.995} C_VEL
LIN {X 0,Y 337.16,Z 185.491,A -85,B 0,C 180,E1 -14360.601,E2 -14360.601} C_VEL
LIN {X 0,Y 334.769,Z 185.789,A -85,B 0,C 180,E1 -14361.901,E2 -14361.901} C_VEL
LIN {X 0,Y 333.746,Z 185.914,A -85,B 0,C 180,E1 -14362.906,E2 -14362.906} C_VEL
LIN {X 0,Y 333.663,Z 185.922,A -85,B 0,C 180,E1 -14363.247,E2 -14363.247} C_VEL
LIN {X 0,Y 333.638,Z 185.926,A -85,B 0,C 180,E1 -14366.792,E2 -14366.792} C_VEL
LIN {X 0,Y 333.696,Z 185.916,A -85,B 0,C 180,E1 -14369.713,E2 -14369.713} C_VEL
LIN {X 0,Y 333.741,Z 185.915,A -85,B 0,C 180,E1 -14372.401,E2 -14372.401} C_VEL
LIN {X 0,Y 333.728,Z 185.912,A -85,B 0,C 180,E1 -14375.091,E2 -14375.091} C_VEL
LIN {X 0,Y 333.682,Z 185.917,A -85,B 0,C 180,E1 -14379.019,E2 -14379.019} C_VEL
LIN {X 0,Y 333.795,Z 185.905,A -85,B 0,C 180,E1 -14381.589,E2 -14381.589} C_VEL
LIN {X 0,Y 333.81,Z 185.905,A -85,B 0,C 180,E1 -14385.577,E2 -14385.577} C_VEL
LIN {X 0,Y 333.818,Z 185.901,A -85,B 0,C 180,E1 -14389.077,E2 -14389.077} C_VEL
LIN {X 0,Y 333.958,Z 185.883,A -85,B 0,C 180,E1 -14392.746,E2 -14392.746} C_VEL
LIN {X 0,Y 333.795,Z 185.907,A -85,B 0,C 180,E1 -14395.169,E2 -14395.169} C_VEL
LIN {X 0,Y 334.103,Z 185.868,A -85,B 0,C 180,E1 -14397.589,E2 -14397.589} C_VEL
LIN {X 0,Y 334.249,Z 185.847,A -85,B 0,C 180,E1 -14400,E2 -14400} C_VEL
LIN {X 0,Y 334.104,Z 185.865,A -85,B 0,C 180,E1 -14402.411,E2 -14402.411} C_VEL
LIN {X 0,Y 333.991,Z 185.879,A -85,B 0,C 180,E1 -14406.039,E2 -14406.039} C_VEL
LIN {X 0,Y 333.85,Z 185.897,A -85,B 0,C 180,E1 -14409.695,E2 -14409.695} C_VEL
LIN {X 0,Y 333.799,Z 185.904,A -85,B 0,C 180,E1 -14413.391,E2 -14413.391} C_VEL
LIN {X 0,Y 333.748,Z 185.91,A -85,B 0,C 180,E1 -14417.146,E2 -14417.146} C_VEL
LIN {X 0,Y 333.734,Z 185.912,A -85,B 0,C 180,E1 -14419.691,E2 -14419.691} C_VEL
LIN {X 0,Y 333.67,Z 185.92,A -85,B 0,C 180,E1 -14423.59,E2 -14423.59} C_VEL
LIN {X 0,Y 333.736,Z 185.915,A -85,B 0,C 180,E1 -14426.246,E2 -14426.246} C_VEL
LIN {X 0,Y 333.691,Z 185.917,A -85,B 0,C 180,E1 -14428.974,E2 -14428.974} C_VEL
LIN {X 0,Y 333.644,Z 185.923,A -85,B 0,C 180,E1 -14432.587,E2 -14432.587} C_VEL
LIN {X 0,Y 333.675,Z 185.921,A -85,B 0,C 180,E1 -14436.139,E2 -14436.139} C_VEL
LIN {X 0,Y 333.633,Z 185.927,A -85,B 0,C 180,E1 -14439.194,E2 -14439.194} C_VEL
LIN {X 0,Y 333.633,Z 185.926,A -85,B 0,C 180,E1 -14442.5,E2 -14442.5} C_VEL
LIN {X 0,Y 333.669,Z 186.075,A -85,B 0,C 180,E1 -14445.133,E2 -14445.133} C_VEL
LIN {X 0,Y 334.267,Z 189.302,A -85,B 0,C 180,E1 -14447.716,E2 -14447.716} C_VEL
LIN {X 0,Y 334.972,Z 193.686,A -85,B 0,C 180,E1 -14450.992,E2 -14450.992} C_VEL
LIN {X 0,Y 335.338,Z 198.059,A -85,B 0,C 180,E1 -14454.068,E2 -14454.068} C_VEL
LIN {X 0,Y 334.973,Z 202.617,A -85,B 0,C 180,E1 -14457.059,E2 -14457.059} C_VEL
LIN {X 0,Y 334.344,Z 207.859,A -85,B 0,C 180,E1 -14460.397,E2 -14460.397} C_VEL
LIN {X 0,Y 333.785,Z 213.264,A -85,B 0,C 180,E1 -14463.758,E2 -14463.758} C_VEL
LIN {X 0,Y 333.168,Z 220.149,A -85,B 0,C 180,E1 -14467.988,E2 -14467.988} C_VEL
LIN {X 0,Y 333.161,Z 220.539,A -85,B 0,C 180,E1 -14468.153,E2 -14468.153} C_VEL
LIN {X 0,Y 335.971,Z 233.418,A -85,B 0,C 180,E1 -14468.837,E2 -14468.837} C_VEL
LIN {X 0,Y 338.054,Z 246.069,A -85,B 0,C 180,E1 -14469.713,E2 -14469.713} C_VEL
LIN {X 0,Y 339.418,Z 258.807,A -85,B 0,C 180,E1 -14470.809,E2 -14470.809} C_VEL
LIN {X 0,Y 338.808,Z 266.632,A -85,B 0,C 180,E1 -14471.558,E2 -14471.558} C_VEL
LIN {X 0,Y 337.37,Z 278.176,A -85,B 0,C 180,E1 -14472.887,E2 -14472.887} C_VEL
LIN {X 0,Y 336.282,Z 287.481,A -85,B 0,C 180,E1 -14474.235,E2 -14474.235} C_VEL
LIN {X 0,Y 335.215,Z 295.965,A -85,B 0,C 180,E1 -14475.738,E2 -14475.738} C_VEL
LIN {X 0,Y 334.021,Z 304.243,A -85,B 0,C 180,E1 -14477.545,E2 -14477.545} C_VEL
LIN {X 0,Y 333.215,Z 310.921,A -85,B 0,C 180,E1 -14479.365,E2 -14479.365} C_VEL
LIN {X 0,Y 332.558,Z 317.034,A -85,B 0,C 180,E1 -14481.493,E2 -14481.493} C_VEL
LIN {X 0,Y 332.179,Z 321.007,A -85,B 0,C 180,E1 -14483.317,E2 -14483.317} C_VEL
LIN {X 0,Y 332.02,Z 323.945,A -85,B 0,C 180,E1 -14485.143,E2 -14485.143} C_VEL
LIN {X 0,Y 332.004,Z 325.345,A -85,B 0,C 180,E1 -14486.359,E2 -14486.359} C_VEL
LIN {X 0,Y 331.905,Z 326.951,A -85,B 0,C 180,E1 -14488.786,E2 -14488.786} C_VEL
LIN {X 0,Y 331.928,Z 327.167,A -85,B 0,C 180,E1 -14490,E2 -14490} C_VEL
LIN {X 0,Y 331.905,Z 326.948,A -85,B 0,C 180,E1 -14491.213,E2 -14491.213} C_VEL
LIN {X 0,Y 332.004,Z 325.341,A -85,B 0,C 180,E1 -14493.641,E2 -14493.641} C_VEL
LIN {X 0,Y 332.073,Z 322.386,A -85,B 0,C 180,E1 -14495.894,E2 -14495.894} C_VEL
LIN {X 0,Y 332.39,Z 318.449,A -85,B 0,C 180,E1 -14497.899,E2 -14497.899} C_VEL
LIN {X 0,Y 332.892,Z 313.718,A -85,B 0,C 180,E1 -14499.723,E2 -14499.723} C_VEL
LIN {X 0,Y 333.695,Z 306.612,A -85,B 0,C 180,E1 -14501.849,E2 -14501.849} C_VEL
LIN {X 0,Y 334.776,Z 298.907,A -85,B 0,C 180,E1 -14503.66,E2 -14503.66} C_VEL
LIN {X 0,Y 336.056,Z 289.231,A -85,B 0,C 180,E1 -14505.464,E2 -14505.464} C_VEL
LIN {X 0,Y 337.223,Z 279.248,A -85,B 0,C 180,E1 -14506.964,E2 -14506.964} C_VEL
LIN {X 0,Y 338.617,Z 267.981,A -85,B 0,C 180,E1 -14508.295,E2 -14508.295} C_VEL
LIN {X 0,Y 339.449,Z 260.409,A -85,B 0,C 180,E1 -14509.031,E2 -14509.031} C_VEL
LIN {X 0,Y 338.445,Z 249.526,A -85,B 0,C 180,E1 -14510.01,E2 -14510.01} C_VEL
LIN {X 0,Y 336.929,Z 238.728,A -85,B 0,C 180,E1 -14510.811,E2 -14510.811} C_VEL
LIN {X 0,Y 334.414,Z 225.954,A -85,B 0,C 180,E1 -14511.571,E2 -14511.571} C_VEL
LIN {X 0,Y 333.158,Z 220.354,A -85,B 0,C 180,E1 -14511.876,E2 -14511.876} C_VEL
LIN {X 0,Y 333.607,Z 215.173,A -85,B 0,C 180,E1 -14515.059,E2 -14515.059} C_VEL
LIN {X 0,Y 334.217,Z 208.932,A -85,B 0,C 180,E1 -14518.924,E2 -14518.924} C_VEL
LIN {X 0,Y 334.863,Z 203.59,A -85,B 0,C 180,E1 -14522.297,E2 -14522.297} C_VEL
LIN {X 0,Y 335.316,Z 199.147,A -85,B 0,C 180,E1 -14525.173,E2 -14525.173} C_VEL
LIN {X 0,Y 335.152,Z 194.741,A -85,B 0,C 180,E1 -14528.214,E2 -14528.214} C_VEL
LIN {X 0,Y 334.593,Z 191.125,A -85,B 0,C 180,E1 -14530.872,E2 -14530.872} C_VEL
LIN {X 0,Y 333.691,Z 186.286,A -85,B 0,C 180,E1 -14534.671,E2 -14534.671} C_VEL
LIN {X 0,Y 333.631,Z 185.932,A -85,B 0,C 180,E1 -14535.061,E2 -14535.061} C_VEL
LIN {X 0,Y 333.64,Z 185.926,A -85,B 0,C 180,E1 -14537.618,E2 -14537.618} C_VEL
LIN {X 0,Y 333.638,Z 185.924,A -85,B 0,C 180,E1 -14541.205,E2 -14541.205} C_VEL
LIN {X 0,Y 333.673,Z 185.921,A -85,B 0,C 180,E1 -14543.861,E2 -14543.861} C_VEL
LIN {X 0,Y 333.642,Z 185.923,A -85,B 0,C 180,E1 -14547.413,E2 -14547.413} C_VEL
LIN {X 0,Y 333.688,Z 185.917,A -85,B 0,C 180,E1 -14551.026,E2 -14551.026} C_VEL
LIN {X 0,Y 333.733,Z 185.915,A -85,B 0,C 180,E1 -14553.753,E2 -14553.753} C_VEL
LIN {X 0,Y 333.655,Z 185.926,A -85,B 0,C 180,E1 -14557.719,E2 -14557.719} C_VEL
LIN {X 0,Y 333.793,Z 185.909,A -85,B 0,C 180,E1 -14561.589,E2 -14561.589} C_VEL
LIN {X 0,Y 333.806,Z 185.906,A -85,B 0,C 180,E1 -14565.576,E2 -14565.576} C_VEL
LIN {X 0,Y 333.815,Z 185.904,A -85,B 0,C 180,E1 -14569.077,E2 -14569.077} C_VEL
LIN {X 0,Y 333.954,Z 185.885,A -85,B 0,C 180,E1 -14572.746,E2 -14572.746} C_VEL
LIN {X 0,Y 333.795,Z 185.908,A -85,B 0,C 180,E1 -14575.169,E2 -14575.169} C_VEL
LIN {X 0,Y 334.101,Z 185.866,A -85,B 0,C 180,E1 -14577.589,E2 -14577.589} C_VEL
LIN {X 0,Y 334.245,Z 185.847,A -85,B 0,C 180,E1 -14580,E2 -14580} C_VEL
LIN {X 0,Y 334.101,Z 185.868,A -85,B 0,C 180,E1 -14582.411,E2 -14582.411} C_VEL
LIN {X 0,Y 333.955,Z 185.882,A -85,B 0,C 180,E1 -14586.565,E2 -14586.565} C_VEL
LIN {X 0,Y 333.818,Z 185.901,A -85,B 0,C 180,E1 -14589.696,E2 -14589.696} C_VEL
LIN {X 0,Y 333.795,Z 185.903,A -85,B 0,C 180,E1 -14593.392,E2 -14593.392} C_VEL
LIN {X 0,Y 333.745,Z 185.91,A -85,B 0,C 180,E1 -14597.146,E2 -14597.146} C_VEL
LIN {X 0,Y 333.738,Z 185.913,A -85,B 0,C 180,E1 -14599.69,E2 -14599.69} C_VEL
LIN {X 0,Y 333.691,Z 185.919,A -85,B 0,C 180,E1 -14602.278,E2 -14602.278} C_VEL
LIN {X 0,Y 333.733,Z 185.913,A -85,B 0,C 180,E1 -14606.247,E2 -14606.247} C_VEL
LIN {X 0,Y 333.703,Z 185.915,A -85,B 0,C 180,E1 -14610.291,E2 -14610.291} C_VEL
LIN {X 0,Y 333.672,Z 185.919,A -85,B 0,C 180,E1 -14614.659,E2 -14614.659} C_VEL
LIN {X 0,Y 333.642,Z 185.925,A -85,B 0,C 180,E1 -14617.653,E2 -14617.653} C_VEL
LIN {X 0,Y 333.642,Z 185.925,A -85,B 0,C 180,E1 -14620.768,E2 -14620.768} C_VEL
LIN {X 0,Y 333.593,Z 185.929,A -85,B 0,C 180,E1 -14624.251,E2 -14624.251} C_VEL
LIN {X 0,Y 333.641,Z 185.924,A -85,B 0,C 180,E1 -14627.619,E2 -14627.619} C_VEL
LIN {X 0,Y 333.645,Z 185.925,A -85,B 0,C 180,E1 -14631.204,E2 -14631.204} C_VEL
LIN {X 0,Y 333.633,Z 185.928,A -85,B 0,C 180,E1 -14632.347,E2 -14632.347} C_VEL
LIN {X 0,Y 333.652,Z 188.72,A -85,B 0,C 180,E1 -14635.339,E2 -14635.339} C_VEL
LIN {X 0,Y 333.498,Z 191.681,A -85,B 0,C 180,E1 -14638.208,E2 -14638.208} C_VEL
LIN {X 0,Y 333.319,Z 194.668,A -85,B 0,C 180,E1 -14640.991,E2 -14640.991} C_VEL
LIN {X 0,Y 333.099,Z 197.673,A -85,B 0,C 180,E1 -14643.7,E2 -14643.7} C_VEL
LIN {X 0,Y 332.855,Z 202.259,A -85,B 0,C 180,E1 -14647.663,E2 -14647.663} C_VEL
LIN {X 0,Y 332.83,Z 202.906,A -85,B 0,C 180,E1 -14648.214,E2 -14648.214} C_VEL
LIN {X 0,Y 336.436,Z 216.215,A -85,B 0,C 180,E1 -14649.013,E2 -14649.013} C_VEL
LIN {X 0,Y 339.09,Z 228.345,A -85,B 0,C 180,E1 -14649.931,E2 -14649.931} C_VEL
LIN {X 0,Y 340.407,Z 237.129,A -85,B 0,C 180,E1 -14650.711,E2 -14650.711} C_VEL
LIN {X 0,Y 339.306,Z 248.22,A -85,B 0,C 180,E1 -14651.743,E2 -14651.743} C_VEL
LIN {X 0,Y 338.053,Z 259.52,A -85,B 0,C 180,E1 -14653.079,E2 -14653.079} C_VEL
LIN {X 0,Y 336.872,Z 269.486,A -85,B 0,C 180,E1 -14654.574,E2 -14654.574} C_VEL
LIN {X 0,Y 335.528,Z 279.125,A -85,B 0,C 180,E1 -14656.371,E2 -14656.371} C_VEL
LIN {X 0,Y 334.448,Z 286.81,A -85,B 0,C 180,E1 -14658.178,E2 -14658.178} C_VEL
LIN {X 0,Y 333.704,Z 292.056,A -85,B 0,C 180,E1 -14659.688,E2 -14659.688} C_VEL
LIN {X 0,Y 333.026,Z 297.143,A -85,B 0,C 180,E1 -14661.505,E2 -14661.505} C_VEL
LIN {X 0,Y 332.661,Z 300.833,A -85,B 0,C 180,E1 -14663.196,E2 -14663.196} C_VEL
LIN {X 0,Y 332.342,Z 304.005,A -85,B 0,C 180,E1 -14665.148,E2 -14665.148} C_VEL
LIN {X 0,Y 332.142,Z 305.403,A -85,B 0,C 180,E1 -14666.361,E2 -14666.361} C_VEL
LIN {X 0,Y 331.984,Z 307.008,A -85,B 0,C 180,E1 -14668.787,E2 -14668.787} C_VEL
LIN {X 0,Y 331.978,Z 307.239,A -85,B 0,C 180,E1 -14670,E2 -14670} C_VEL
LIN {X 0,Y 331.984,Z 307.049,A -85,B 0,C 180,E1 -14671.213,E2 -14671.213} C_VEL
LIN {X 0,Y 332.141,Z 305.497,A -85,B 0,C 180,E1 -14673.64,E2 -14673.64} C_VEL
LIN {X 0,Y 332.316,Z 304.139,A -85,B 0,C 180,E1 -14674.853,E2 -14674.853} C_VEL
LIN {X 0,Y 332.658,Z 301.046,A -85,B 0,C 180,E1 -14676.801,E2 -14676.801} C_VEL
LIN {X 0,Y 333.024,Z 297.39,A -85,B 0,C 180,E1 -14678.495,E2 -14678.495} C_VEL
LIN {X 0,Y 333.67,Z 292.375,A -85,B 0,C 180,E1 -14680.314,E2 -14680.314} C_VEL
LIN {X 0,Y 334.558,Z 286.06,A -85,B 0,C 180,E1 -14682.127,E2 -14682.127} C_VEL
LIN {X 0,Y 335.678,Z 278.153,A -85,B 0,C 180,E1 -14683.932,E2 -14683.932} C_VEL
LIN {X 0,Y 337.097,Z 268.315,A -85,B 0,C 180,E1 -14685.726,E2 -14685.726} C_VEL
LIN {X 0,Y 338.206,Z 258.436,A -85,B 0,C 180,E1 -14687.166,E2 -14687.166} C_VEL
LIN {X 0,Y 339.368,Z 247.763,A -85,B 0,C 180,E1 -14688.41,E2 -14688.41} C_VEL
LIN {X 0,Y 340.475,Z 236.523,A -85,B 0,C 180,E1 -14689.446,E2 -14689.446} C_VEL
LIN {X 0,Y 338.462,Z 224.911,A -85,B 0,C 180,E1 -14690.458,E2 -14690.458} C_VEL
LIN {X 0,Y 335.337,Z 211.96,A -85,B 0,C 180,E1 -14691.374,E2 -14691.374} C_VEL
LIN {X 0,Y 332.809,Z 202.882,A -85,B 0,C 180,E1 -14691.919,E2 -14691.919} C_VEL
LIN {X 0,Y 333,Z 199.311,A -85,B 0,C 180,E1 -14694.968,E2 -14694.968} C_VEL
LIN {X 0,Y 333.239,Z 196.307,A -85,B 0,C 180,E1 -14697.652,E2 -14697.652} C_VEL
LIN {X 0,Y 333.412,Z 193.311,A -85,B 0,C 180,E1 -14700.391,E2 -14700.391} C_VEL
LIN {X 0,Y 333.597,Z 190.327,A -85,B 0,C 180,E1 -14703.213,E2 -14703.213} C_VEL
LIN {X 0,Y 333.714,Z 187.355,A -85,B 0,C 180,E1 -14706.134,E2 -14706.134} C_VEL
LIN {X 0,Y 333.613,Z 185.931,A -85,B 0,C 180,E1 -14707.656,E2 -14707.656} C_VEL
LIN {X 0,Y 333.605,Z 185.928,A -85,B 0,C 180,E1 -14710.774,E2 -14710.774} C_VEL
LIN {X 0,Y 333.594,Z 185.928,A -85,B 0,C 180,E1 -14714.25,E2 -14714.25} C_VEL
LIN {X 0,Y 333.619,Z 185.924,A -85,B 0,C 180,E1 -14718,E2 -14718} C_VEL
LIN {X 0,Y 333.641,Z 185.925,A -85,B 0,C 180,E1 -14721.205,E2 -14721.205} C_VEL
LIN {X 0,Y 333.663,Z 185.922,A -85,B 0,C 180,E1 -14723.247,E2 -14723.247} C_VEL
LIN {X 0,Y 332.986,Z 186.008,A -85,B 0,C 180,E1 -14724.255,E2 -14724.255} C_VEL
LIN {X 0,Y 330.102,Z 186.364,A -85,B 0,C 180,E1 -14725.893,E2 -14725.893} C_VEL
LIN {X 0,Y 327.673,Z 186.666,A -85,B 0,C 180,E1 -14727.221,E2 -14727.221} C_VEL
LIN {X 0,Y 326.65,Z 186.796,A -85,B 0,C 180,E1 -14728.249,E2 -14728.249} C_VEL
LIN {X 0,Y 326.577,Z 186.802,A -85,B 0,C 180,E1 -14728.597,E2 -14728.597} C_VEL
LIN {X 0,Y 326.658,Z 186.794,A -85,B 0,C 180,E1 -14731.898,E2 -14731.898} C_VEL
LIN {X 0,Y 326.69,Z 186.791,A -85,B 0,C 180,E1 -14734.627,E2 -14734.627} C_VEL
LIN {X 0,Y 326.647,Z 186.795,A -85,B 0,C 180,E1 -14738.545,E2 -14738.545} C_VEL
LIN {X 0,Y 326.746,Z 186.781,A -85,B 0,C 180,E1 -14741.177,E2 -14741.177} C_VEL
LIN {X 0,Y 326.765,Z 186.781,A -85,B 0,C 180,E1 -14745.433,E2 -14745.433} C_VEL
LIN {X 0,Y 326.759,Z 186.78,A -85,B 0,C 180,E1 -14748.838,E2 -14748.838} C_VEL
LIN {X 0,Y 326.914,Z 186.76,A -85,B 0,C 180,E1 -14752.589,E2 -14752.589} C_VEL
LIN {X 0,Y 326.762,Z 186.782,A -85,B 0,C 180,E1 -14755.065,E2 -14755.065} C_VEL
LIN {X 0,Y 327.043,Z 186.748,A -85,B 0,C 180,E1 -14757.537,E2 -14757.537} C_VEL
LIN {X 0,Y 327.2,Z 186.725,A -85,B 0,C 180,E1 -14760,E2 -14760} C_VEL
LIN {X 0,Y 327.044,Z 186.745,A -85,B 0,C 180,E1 -14762.463,E2 -14762.463} C_VEL
LIN {X 0,Y 326.945,Z 186.757,A -85,B 0,C 180,E1 -14766.17,E2 -14766.17} C_VEL
LIN {X 0,Y 326.806,Z 186.774,A -85,B 0,C 180,E1 -14769.906,E2 -14769.906} C_VEL
LIN {X 0,Y 326.761,Z 186.78,A -85,B 0,C 180,E1 -14773.685,E2 -14773.685} C_VEL
LIN {X 0,Y 326.7,Z 186.788,A -85,B 0,C 180,E1 -14777.528,E2 -14777.528} C_VEL
LIN {X 0,Y 326.66,Z 186.796,A -85,B 0,C 180,E1 -14780.135,E2 -14780.135} C_VEL
LIN {X 0,Y 326.65,Z 186.798,A -85,B 0,C 180,E1 -14784.129,E2 -14784.129} C_VEL
LIN {X 0,Y 326.684,Z 186.79,A -85,B 0,C 180,E1 -14786.858,E2 -14786.858} C_VEL
LIN {X 0,Y 326.635,Z 186.797,A -85,B 0,C 180,E1 -14790.61,E2 -14790.61} C_VEL
LIN {X 0,Y 326.608,Z 186.803,A -85,B 0,C 180,E1 -14794.019,E2 -14794.019} C_VEL
LIN {X 0,Y 326.624,Z 186.8,A -85,B 0,C 180,E1 -14797.237,E2 -14797.237} C_VEL
LIN {X 0,Y 326.577,Z 186.807,A -85,B 0,C 180,E1 -14801.131,E2 -14801.131} C_VEL
LIN {X 0,Y 326.617,Z 186.989,A -85,B 0,C 180,E1 -14804.758,E2 -14804.758} C_VEL
LIN {X 0,Y 327.495,Z 191.833,A -85,B 0,C 180,E1 -14808.686,E2 -14808.686} C_VEL
LIN {X 0,Y 328.109,Z 195.717,A -85,B 0,C 180,E1 -14811.598,E2 -14811.598} C_VEL
LIN {X 0,Y 328.292,Z 200.081,A -85,B 0,C 180,E1 -14814.689,E2 -14814.689} C_VEL
LIN {X 0,Y 327.716,Z 205.52,A -85,B 0,C 180,E1 -14818.304,E2 -14818.304} C_VEL
LIN {X 0,Y 326.945,Z 211.988,A -85,B 0,C 180,E1 -14822.473,E2 -14822.473} C_VEL
LIN {X 0,Y 326.288,Z 218.384,A -85,B 0,C 180,E1 -14826.517,E2 -14826.517} C_VEL
LIN {X 0,Y 326.163,Z 220.192,A -85,B 0,C 180,E1 -14827.649,E2 -14827.649} C_VEL
LIN {X 0,Y 329.188,Z 234.039,A -85,B 0,C 180,E1 -14828.423,E2 -14828.423} C_VEL
LIN {X 0,Y 331.307,Z 247.055,A -85,B 0,C 180,E1 -14829.366,E2 -14829.366} C_VEL
LIN {X 0,Y 332.515,Z 258.593,A -85,B 0,C 180,E1 -14830.395,E2 -14830.395} C_VEL
LIN {X 0,Y 332.443,Z 263.46,A -85,B 0,C 180,E1 -14830.872,E2 -14830.872} C_VEL
LIN {X 0,Y 331.061,Z 274.434,A -85,B 0,C 180,E1 -14832.072,E2 -14832.072} C_VEL
LIN {X 0,Y 329.7,Z 284.811,A -85,B 0,C 180,E1 -14833.511,E2 -14833.511} C_VEL
LIN {X 0,Y 328.478,Z 294.167,A -85,B 0,C 180,E1 -14835.123,E2 -14835.123} C_VEL
LIN {X 0,Y 327.265,Z 302.795,A -85,B 0,C 180,E1 -14836.968,E2 -14836.968} C_VEL
LIN {X 0,Y 326.346,Z 309.695,A -85,B 0,C 180,E1 -14838.824,E2 -14838.824} C_VEL
LIN {X 0,Y 325.674,Z 315.227,A -85,B 0,C 180,E1 -14840.686,E2 -14840.686} C_VEL
LIN {X 0,Y 325.212,Z 319.568,A -85,B 0,C 180,E1 -14842.55,E2 -14842.55} C_VEL
LIN {X 0,Y 324.996,Z 322.418,A -85,B 0,C 180,E1 -14844.125,E2 -14844.125} C_VEL
LIN {X 0,Y 324.91,Z 325.132,A -85,B 0,C 180,E1 -14846.279,E2 -14846.279} C_VEL
LIN {X 0,Y 324.814,Z 326.738,A -85,B 0,C 180,E1 -14848.76,E2 -14848.76} C_VEL
LIN {X 0,Y 324.835,Z 326.954,A -85,B 0,C 180,E1 -14850,E2 -14850} C_VEL
LIN {X 0,Y 324.814,Z 326.735,A -85,B 0,C 180,E1 -14851.239,E2 -14851.239} C_VEL
LIN {X 0,Y 324.91,Z 325.128,A -85,B 0,C 180,E1 -14853.72,E2 -14853.72} C_VEL
LIN {X 0,Y 324.996,Z 322.408,A -85,B 0,C 180,E1 -14855.875,E2 -14855.875} C_VEL
LIN {X 0,Y 325.344,Z 318.234,A -85,B 0,C 180,E1 -14858.071,E2 -14858.071} C_VEL
LIN {X 0,Y 325.873,Z 313.503,A -85,B 0,C 180,E1 -14859.935,E2 -14859.935} C_VEL
LIN {X 0,Y 326.724,Z 306.397,A -85,B 0,C 180,E1 -14862.106,E2 -14862.106} C_VEL
LIN {X 0,Y 327.865,Z 298.691,A -85,B 0,C 180,E1 -14863.954,E2 -14863.954} C_VEL
LIN {X 0,Y 328.947,Z 290.803,A -85,B 0,C 180,E1 -14865.489,E2 -14865.489} C_VEL
LIN {X 0,Y 330.255,Z 280.211,A -85,B 0,C 180,E1 -14867.157,E2 -14867.157} C_VEL
LIN {X 0,Y 331.675,Z 269.187,A -85,B 0,C 180,E1 -14868.532,E2 -14868.532} C_VEL
LIN {X 0,Y 332.574,Z 260.185,A -85,B 0,C 180,E1 -14869.44,E2 -14869.44} C_VEL
LIN {X 0,Y 331.478,Z 248.504,A -85,B 0,C 180,E1 -14870.507,E2 -14870.507} C_VEL
LIN {X 0,Y 329.5,Z 235.892,A -85,B 0,C 180,E1 -14871.443,E2 -14871.443} C_VEL
LIN {X 0,Y 326.738,Z 222.933,A -85,B 0,C 180,E1 -14872.204,E2 -14872.204} C_VEL
LIN {X 0,Y 326.154,Z 220.131,A -85,B 0,C 180,E1 -14872.378,E2 -14872.378} C_VEL
LIN {X 0,Y 326.694,Z 214.122,A -85,B 0,C 180,E1 -14876.168,E2 -14876.168} C_VEL
LIN {X 0,Y 327.287,Z 208.742,A -85,B 0,C 180,E1 -14879.596,E2 -14879.596} C_VEL
LIN {X 0,Y 327.998,Z 203.025,A -85,B 0,C 180,E1 -14883.316,E2 -14883.316} C_VEL
LIN {X 0,Y 328.3,Z 199.666,A -85,B 0,C 180,E1 -14885.563,E2 -14885.563} C_VEL
LIN {X 0,Y 328.132,Z 195.652,A -85,B 0,C 180,E1 -14888.398,E2 -14888.398} C_VEL
LIN {X 0,Y 327.399,Z 191.293,A -85,B 0,C 180,E1 -14891.716,E2 -14891.716} C_VEL
LIN {X 0,Y 326.575,Z 186.81,A -85,B 0,C 180,E1 -14895.448,E2 -14895.448} C_VEL
LIN {X 0,Y 326.574,Z 186.808,A -85,B 0,C 180,E1 -14898.869,E2 -14898.869} C_VEL
LIN {X 0,Y 326.621,Z 186.8,A -85,B 0,C 180,E1 -14902.762,E2 -14902.762} C_VEL
LIN {X 0,Y 326.605,Z 186.802,A -85,B 0,C 180,E1 -14905.98,E2 -14905.98} C_VEL
LIN {X 0,Y 326.646,Z 186.797,A -85,B 0,C 180,E1 -14910.339,E2 -14910.339} C_VEL
LIN {X 0,Y 326.688,Z 186.79,A -85,B 0,C 180,E1 -14914.516,E2 -14914.516} C_VEL
LIN {X 0,Y 326.618,Z 186.798,A -85,B 0,C 180,E1 -14918.543,E2 -14918.543} C_VEL
LIN {X 0,Y 326.742,Z 186.784,A -85,B 0,C 180,E1 -14921.177,E2 -14921.177} C_VEL
LIN {X 0,Y 326.761,Z 186.785,A -85,B 0,C 180,E1 -14925.433,E2 -14925.433} C_VEL
LIN {X 0,Y 326.755,Z 186.781,A -85,B 0,C 180,E1 -14928.838,E2 -14928.838} C_VEL
LIN {X 0,Y 326.911,Z 186.762,A -85,B 0,C 180,E1 -14932.589,E2 -14932.589} C_VEL
LIN {X 0,Y 326.762,Z 186.784,A -85,B 0,C 180,E1 -14935.065,E2 -14935.065} C_VEL
LIN {X 0,Y 327.042,Z 186.745,A -85,B 0,C 180,E1 -14937.537,E2 -14937.537} C_VEL
LIN {X 0,Y 327.197,Z 186.725,A -85,B 0,C 180,E1 -14940,E2 -14940} C_VEL
LIN {X 0,Y 327.041,Z 186.747,A -85,B 0,C 180,E1 -14942.463,E2 -14942.463} C_VEL
LIN {X 0,Y 326.916,Z 186.76,A -85,B 0,C 180,E1 -14946.554,E2 -14946.554} C_VEL
LIN {X 0,Y 326.78,Z 186.778,A -85,B 0,C 180,E1 -14949.907,E2 -14949.907} C_VEL
LIN {X 0,Y 326.757,Z 186.781,A -85,B 0,C 180,E1 -14953.686,E2 -14953.686} C_VEL
LIN {X 0,Y 326.698,Z 186.789,A -85,B 0,C 180,E1 -14957.528,E2 -14957.528} C_VEL
LIN {X 0,Y 326.663,Z 186.796,A -85,B 0,C 180,E1 -14960.135,E2 -14960.135} C_VEL
LIN {X 0,Y 326.65,Z 186.796,A -85,B 0,C 180,E1 -14964.129,E2 -14964.129} C_VEL
LIN {X 0,Y 326.681,Z 186.79,A -85,B 0,C 180,E1 -14966.858,E2 -14966.858} C_VEL
LIN {X 0,Y 326.638,Z 186.795,A -85,B 0,C 180,E1 -14970.612,E2 -14970.612} C_VEL
LIN {X 0,Y 326.605,Z 186.8,A -85,B 0,C 180,E1 -14974.02,E2 -14974.02} C_VEL
LIN {X 0,Y 326.622,Z 186.802,A -85,B 0,C 180,E1 -14977.238,E2 -14977.238} C_VEL
LIN {X 0,Y 326.575,Z 186.809,A -85,B 0,C 180,E1 -14981.131,E2 -14981.131} C_VEL
LIN {X 0,Y 326.527,Z 186.813,A -85,B 0,C 180,E1 -14984.743,E2 -14984.743} C_VEL
LIN {X 0,Y 326.576,Z 186.804,A -85,B 0,C 180,E1 -14988.155,E2 -14988.155} C_VEL
LIN {X 0,Y 326.589,Z 186.804,A -85,B 0,C 180,E1 -14991.387,E2 -14991.387} C_VEL
LIN {X 0,Y 326.608,Z 187.408,A -85,B 0,C 180,E1 -14992.951,E2 -14992.951} C_VEL
LIN {X 0,Y 326.574,Z 190.389,A -85,B 0,C 180,E1 -14995.977,E2 -14995.977} C_VEL
LIN {X 0,Y 326.372,Z 193.976,A -85,B 0,C 180,E1 -14999.469,E2 -14999.469} C_VEL
LIN {X 0,Y 326.09,Z 197.878,A -85,B 0,C 180,E1 -15003.09,E2 -15003.09} C_VEL
LIN {X 0,Y 325.825,Z 202.464,A -85,B 0,C 180,E1 -15007.154,E2 -15007.154} C_VEL
LIN {X 0,Y 325.808,Z 203.111,A -85,B 0,C 180,E1 -15007.715,E2 -15007.715} C_VEL
LIN {X 0,Y 329.593,Z 216.825,A -85,B 0,C 180,E1 -15008.576,E2 -15008.576} C_VEL
LIN {X 0,Y 332.287,Z 229.127,A -85,B 0,C 180,E1 -15009.542,E2 -15009.542} C_VEL
LIN {X 0,Y 333.61,Z 237.352,A -85,B 0,C 180,E1 -15010.302,E2 -15010.302} C_VEL
LIN {X 0,Y 332.57,Z 248.438,A -85,B 0,C 180,E1 -15011.36,E2 -15011.36} C_VEL
LIN {X 0,Y 331.252,Z 259.738,A -85,B 0,C 180,E1 -15012.721,E2 -15012.721} C_VEL
LIN {X 0,Y 330.044,Z 269.702,A -85,B 0,C 180,E1 -15014.247,E2 -15014.247} C_VEL
LIN {X 0,Y 328.642,Z 279.341,A -85,B 0,C 180,E1 -15016.08,E2 -15016.08} C_VEL
LIN {X 0,Y 327.505,Z 287.025,A -85,B 0,C 180,E1 -15017.923,E2 -15017.923} C_VEL
LIN {X 0,Y 326.431,Z 294.079,A -85,B 0,C 180,E1 -15020.082,E2 -15020.082} C_VEL
LIN {X 0,Y 325.845,Z 298.773,A -85,B 0,C 180,E1 -15021.941,E2 -15021.941} C_VEL
LIN {X 0,Y 325.449,Z 302.364,A -85,B 0,C 180,E1 -15023.802,E2 -15023.802} C_VEL
LIN {X 0,Y 325.265,Z 304.219,A -85,B 0,C 180,E1 -15025.042,E2 -15025.042} C_VEL
LIN {X 0,Y 325.075,Z 305.617,A -85,B 0,C 180,E1 -15026.282,E2 -15026.282} C_VEL
LIN {X 0,Y 324.891,Z 307.221,A -85,B 0,C 180,E1 -15028.761,E2 -15028.761} C_VEL
LIN {X 0,Y 324.883,Z 307.452,A -85,B 0,C 180,E1 -15030,E2 -15030} C_VEL
LIN {X 0,Y 324.891,Z 307.261,A -85,B 0,C 180,E1 -15031.24,E2 -15031.24} C_VEL
LIN {X 0,Y 325.073,Z 305.709,A -85,B 0,C 180,E1 -15033.719,E2 -15033.719} C_VEL
LIN {X 0,Y 325.241,Z 304.352,A -85,B 0,C 180,E1 -15034.959,E2 -15034.959} C_VEL
LIN {X 0,Y 325.551,Z 301.592,A -85,B 0,C 180,E1 -15036.757,E2 -15036.757} C_VEL
LIN {X 0,Y 325.982,Z 297.602,A -85,B 0,C 180,E1 -15038.68,E2 -15038.68} C_VEL
LIN {X 0,Y 326.686,Z 292.587,A -85,B 0,C 180,E1 -15040.537,E2 -15040.537} C_VEL
LIN {X 0,Y 327.626,Z 286.27,A -85,B 0,C 180,E1 -15042.387,E2 -15042.387} C_VEL
LIN {X 0,Y 328.77,Z 278.364,A -85,B 0,C 180,E1 -15044.231,E2 -15044.231} C_VEL
LIN {X 0,Y 330.28,Z 268.524,A -85,B 0,C 180,E1 -15046.059,E2 -15046.059} C_VEL
LIN {X 0,Y 331.453,Z 258.201,A -85,B 0,C 180,E1 -15047.587,E2 -15047.587} C_VEL
LIN {X 0,Y 332.642,Z 247.97,A -85,B 0,C 180,E1 -15048.796,E2 -15048.796} C_VEL
LIN {X 0,Y 333.67,Z 238.531,A -85,B 0,C 180,E1 -15049.695,E2 -15049.695} C_VEL
LIN {X 0,Y 332.283,Z 229.029,A -85,B 0,C 180,E1 -15050.575,E2 -15050.575} C_VEL
LIN {X 0,Y 329.459,Z 216.276,A -85,B 0,C 180,E1 -15051.573,E2 -15051.573} C_VEL
LIN {X 0,Y 325.796,Z 203.097,A -85,B 0,C 180,E1 -15052.411,E2 -15052.411} C_VEL
LIN {X 0,Y 325.968,Z 199.517,A -85,B 0,C 180,E1 -15055.544,E2 -15055.544} C_VEL
LIN {X 0,Y 326.228,Z 196.508,A -85,B 0,C 180,E1 -15058.291,E2 -15058.291} C_VEL
LIN {X 0,Y 326.423,Z 193.495,A -85,B 0,C 180,E1 -15061.113,E2 -15061.113} C_VEL
LIN {X 0,Y 326.61,Z 190.506,A -85,B 0,C 180,E1 -15064.019,E2 -15064.019} C_VEL
LIN {X 0,Y 326.604,Z 187.341,A -85,B 0,C 180,E1 -15067.233,E2 -15067.233} C_VEL
LIN {X 0,Y 326.569,Z 186.808,A -85,B 0,C 180,E1 -15069.218,E2 -15069.218} C_VEL
LIN {X 0,Y 326.575,Z 186.805,A -85,B 0,C 180,E1 -15072.971,E2 -15072.971} C_VEL
LIN {X 0,Y 326.577,Z 186.807,A -85,B 0,C 180,E1 -15077.028,E2 -15077.028} C_VEL
LIN {X 0,Y 326.6,Z 186.805,A -85,B 0,C 180,E1 -15080.776,E2 -15080.776} C_VEL
LIN {X 0,Y 326.613,Z 186.802,A -85,B 0,C 180,E1 -15084.48,E2 -15084.48} C_VEL
LIN {X 0,Y 326.609,Z 186.798,A -85,B 0,C 180,E1 -15087.455,E2 -15087.455} C_VEL
LIN {X 0,Y 326.577,Z 186.802,A -85,B 0,C 180,E1 -15088.597,E2 -15088.597} C_VEL
LIN {X 0,Y 325.946,Z 186.885,A -85,B 0,C 180,E1 -15089.627,E2 -15089.627} C_VEL
LIN {X 0,Y 323.138,Z 187.235,A -85,B 0,C 180,E1 -15091.304,E2 -15091.304} C_VEL
LIN {X 0,Y 320.743,Z 187.532,A -85,B 0,C 180,E1 -15092.662,E2 -15092.662} C_VEL
LIN {X 0,Y 319.716,Z 187.659,A -85,B 0,C 180,E1 -15093.714,E2 -15093.714} C_VEL
LIN {X 0,Y 319.634,Z 187.67,A -85,B 0,C 180,E1 -15094.07,E2 -15094.07} C_VEL
LIN {X 0,Y 319.598,Z 187.675,A -85,B 0,C 180,E1 -15098.048,E2 -15098.048} C_VEL
LIN {X 0,Y 319.69,Z 187.66,A -85,B 0,C 180,E1 -15100.962,E2 -15100.962} C_VEL
LIN {X 0,Y 319.732,Z 187.656,A -85,B 0,C 180,E1 -15105.276,E2 -15105.276} C_VEL
LIN {X 0,Y 319.716,Z 187.657,A -85,B 0,C 180,E1 -15108.589,E2 -15108.589} C_VEL
LIN {X 0,Y 319.854,Z 187.64,A -85,B 0,C 180,E1 -15112.424,E2 -15112.424} C_VEL
LIN {X 0,Y 319.731,Z 187.657,A -85,B 0,C 180,E1 -15114.956,E2 -15114.956} C_VEL
LIN {X 0,Y 319.987,Z 187.627,A -85,B 0,C 180,E1 -15117.482,E2 -15117.482} C_VEL
LIN {X 0,Y 320.152,Z 187.603,A -85,B 0,C 180,E1 -15120,E2 -15120} C_VEL
LIN {X 0,Y 319.988,Z 187.624,A -85,B 0,C 180,E1 -15122.518,E2 -15122.518} C_VEL
LIN {X 0,Y 319.902,Z 187.635,A -85,B 0,C 180,E1 -15126.306,E2 -15126.306} C_VEL
LIN {X 0,Y 319.753,Z 187.654,A -85,B 0,C 180,E1 -15130.127,E2 -15130.127} C_VEL
LIN {X 0,Y 319.732,Z 187.66,A -85,B 0,C 180,E1 -15134.724,E2 -15134.724} C_VEL
LIN {X 0,Y 319.69,Z 187.662,A -85,B 0,C 180,E1 -15139.038,E2 -15139.038} C_VEL
LIN {X 0,Y 319.561,Z 187.677,A -85,B 0,C 180,E1 -15143.32,E2 -15143.32} C_VEL
LIN {X 0,Y 319.635,Z 187.672,A -85,B 0,C 180,E1 -15146.088,E2 -15146.088} C_VEL
LIN {X 0,Y 319.581,Z 187.675,A -85,B 0,C 180,E1 -15148.935,E2 -15148.935} C_VEL
LIN {X 0,Y 319.532,Z 187.686,A -85,B 0,C 180,E1 -15151.862,E2 -15151.862} C_VEL
LIN {X 0,Y 319.58,Z 187.68,A -85,B 0,C 180,E1 -15155.543,E2 -15155.543} C_VEL
LIN {X 0,Y 319.56,Z 187.68,A -85,B 0,C 180,E1 -15159.669,E2 -15159.669} C_VEL
LIN {X 0,Y 319.523,Z 187.685,A -85,B 0,C 180,E1 -15163.461,E2 -15163.461} C_VEL
LIN {X 0,Y 319.548,Z 187.93,A -85,B 0,C 180,E1 -15164.384,E2 -15164.384} C_VEL
LIN {X 0,Y 320.427,Z 192.538,A -85,B 0,C 180,E1 -15168.222,E2 -15168.222} C_VEL
LIN {X 0,Y 320.919,Z 195.511,A -85,B 0,C 180,E1 -15170.573,E2 -15170.573} C_VEL
LIN {X 0,Y 321.235,Z 198.813,A -85,B 0,C 180,E1 -15173.012,E2 -15173.012} C_VEL
LIN {X 0,Y 321.191,Z 202.079,A -85,B 0,C 180,E1 -15175.326,E2 -15175.326} C_VEL
LIN {X 0,Y 320.568,Z 207.158,A -85,B 0,C 180,E1 -15178.762,E2 -15178.762} C_VEL
LIN {X 0,Y 319.867,Z 212.865,A -85,B 0,C 180,E1 -15182.522,E2 -15182.522} C_VEL
LIN {X 0,Y 319.218,Z 219.237,A -85,B 0,C 180,E1 -15186.653,E2 -15186.653} C_VEL
LIN {X 0,Y 319.143,Z 220.098,A -85,B 0,C 180,E1 -15187.139,E2 -15187.139} C_VEL
LIN {X 0,Y 322.09,Z 233.149,A -85,B 0,C 180,E1 -15187.886,E2 -15187.886} C_VEL
LIN {X 0,Y 324.17,Z 245.42,A -85,B 0,C 180,E1 -15188.787,E2 -15188.787} C_VEL
LIN {X 0,Y 325.44,Z 256.598,A -85,B 0,C 180,E1 -15189.786,E2 -15189.786} C_VEL
LIN {X 0,Y 325.722,Z 263.251,A -85,B 0,C 180,E1 -15190.461,E2 -15190.461} C_VEL
LIN {X 0,Y 324.278,Z 274.224,A -85,B 0,C 180,E1 -15191.684,E2 -15191.684} C_VEL
LIN {X 0,Y 322.913,Z 284.229,A -85,B 0,C 180,E1 -15193.093,E2 -15193.093} C_VEL
LIN {X 0,Y 321.578,Z 293.955,A -85,B 0,C 180,E1 -15194.796,E2 -15194.796} C_VEL
LIN {X 0,Y 320.512,Z 301.261,A -85,B 0,C 180,E1 -15196.366,E2 -15196.366} C_VEL
LIN {X 0,Y 319.465,Z 308.457,A -85,B 0,C 180,E1 -15198.258,E2 -15198.258} C_VEL
LIN {X 0,Y 318.648,Z 315.015,A -85,B 0,C 180,E1 -15200.478,E2 -15200.478} C_VEL
LIN {X 0,Y 318.152,Z 319.355,A -85,B 0,C 180,E1 -15202.383,E2 -15202.383} C_VEL
LIN {X 0,Y 317.888,Z 322.501,A -85,B 0,C 180,E1 -15204.201,E2 -15204.201} C_VEL
LIN {X 0,Y 317.819,Z 324.919,A -85,B 0,C 180,E1 -15206.196,E2 -15206.196} C_VEL
LIN {X 0,Y 317.759,Z 325.917,A -85,B 0,C 180,E1 -15207.464,E2 -15207.464} C_VEL
LIN {X 0,Y 317.727,Z 326.525,A -85,B 0,C 180,E1 -15208.732,E2 -15208.732} C_VEL
LIN {X 0,Y 317.744,Z 326.742,A -85,B 0,C 180,E1 -15210,E2 -15210} C_VEL
LIN {X 0,Y 317.727,Z 326.522,A -85,B 0,C 180,E1 -15211.267,E2 -15211.267} C_VEL
LIN {X 0,Y 317.759,Z 325.913,A -85,B 0,C 180,E1 -15212.535,E2 -15212.535} C_VEL
LIN {X 0,Y 317.819,Z 324.914,A -85,B 0,C 180,E1 -15213.803,E2 -15213.803} C_VEL
LIN {X 0,Y 317.9,Z 322.459,A -85,B 0,C 180,E1 -15215.82,E2 -15215.82} C_VEL
LIN {X 0,Y 318.15,Z 319.336,A -85,B 0,C 180,E1 -15217.616,E2 -15217.616} C_VEL
LIN {X 0,Y 318.648,Z 314.988,A -85,B 0,C 180,E1 -15219.521,E2 -15219.521} C_VEL
LIN {X 0,Y 319.327,Z 309.45,A -85,B 0,C 180,E1 -15221.424,E2 -15221.424} C_VEL
LIN {X 0,Y 320.329,Z 302.543,A -85,B 0,C 180,E1 -15223.318,E2 -15223.318} C_VEL
LIN {X 0,Y 321.367,Z 295.492,A -85,B 0,C 180,E1 -15224.889,E2 -15224.889} C_VEL
LIN {X 0,Y 322.649,Z 286.208,A -85,B 0,C 180,E1 -15226.581,E2 -15226.581} C_VEL
LIN {X 0,Y 324.07,Z 275.32,A -85,B 0,C 180,E1 -15228.164,E2 -15228.164} C_VEL
LIN {X 0,Y 325.485,Z 264.687,A -85,B 0,C 180,E1 -15229.389,E2 -15229.389} C_VEL
LIN {X 0,Y 325.667,Z 259.96,A -85,B 0,C 180,E1 -15229.87,E2 -15229.87} C_VEL
LIN {X 0,Y 324.506,Z 247.897,A -85,B 0,C 180,E1 -15230.996,E2 -15230.996} C_VEL
LIN {X 0,Y 322.36,Z 234.578,A -85,B 0,C 180,E1 -15232.002,E2 -15232.002} C_VEL
LIN {X 0,Y 319.64,Z 222.379,A -85,B 0,C 180,E1 -15232.736,E2 -15232.736} C_VEL
LIN {X 0,Y 319.158,Z 219.951,A -85,B 0,C 180,E1 -15232.874,E2 -15232.874} C_VEL
LIN {X 0,Y 319.741,Z 213.919,A -85,B 0,C 180,E1 -15236.781,E2 -15236.781} C_VEL
LIN {X 0,Y 320.351,Z 208.55,A -85,B 0,C 180,E1 -15240.303,E2 -15240.303} C_VEL
LIN {X 0,Y 321.041,Z 203.465,A -85,B 0,C 180,E1 -15243.708,E2 -15243.708} C_VEL
LIN {X 0,Y 321.25,Z 199.861,A -85,B 0,C 180,E1 -15246.205,E2 -15246.205} C_VEL
LIN {X 0,Y 321.155,Z 197.359,A -85,B 0,C 180,E1 -15248.019,E2 -15248.019} C_VEL
LIN {X 0,Y 320.552,Z 193.315,A -85,B 0,C 180,E1 -15251.127,E2 -15251.127} C_VEL
LIN {X 0,Y 319.784,Z 188.985,A -85,B 0,C 180,E1 -15254.69,E2 -15254.69} C_VEL
LIN {X 0,Y 319.528,Z 187.688,A -85,B 0,C 180,E1 -15255.958,E2 -15255.958} C_VEL
LIN {X 0,Y 319.525,Z 187.687,A -85,B 0,C 180,E1 -15258.711,E2 -15258.711} C_VEL
LIN {X 0,Y 319.546,Z 187.683,A -85,B 0,C 180,E1 -15262.351,E2 -15262.351} C_VEL
LIN {X 0,Y 319.558,Z 187.678,A -85,B 0,C 180,E1 -15265.123,E2 -15265.123} C_VEL
LIN {X 0,Y 319.564,Z 187.677,A -85,B 0,C 180,E1 -15269.059,E2 -15269.059} C_VEL
LIN {X 0,Y 319.603,Z 187.673,A -85,B 0,C 180,E1 -15272.498,E2 -15272.498} C_VEL
LIN {X 0,Y 319.601,Z 187.673,A -85,B 0,C 180,E1 -15275.304,E2 -15275.304} C_VEL
LIN {X 0,Y 319.601,Z 187.675,A -85,B 0,C 180,E1 -15279.4,E2 -15279.4} C_VEL
LIN {X 0,Y 319.656,Z 187.667,A -85,B 0,C 180,E1 -15282.073,E2 -15282.073} C_VEL
LIN {X 0,Y 319.73,Z 187.657,A -85,B 0,C 180,E1 -15286.008,E2 -15286.008} C_VEL
LIN {X 0,Y 319.733,Z 187.655,A -85,B 0,C 180,E1 -15289.872,E2 -15289.872} C_VEL
LIN {X 0,Y 319.899,Z 187.636,A -85,B 0,C 180,E1 -15293.694,E2 -15293.694} C_VEL
LIN {X 0,Y 319.985,Z 187.625,A -85,B 0,C 180,E1 -15297.482,E2 -15297.482} C_VEL
LIN {X 0,Y 320.149,Z 187.604,A -85,B 0,C 180,E1 -15300,E2 -15300} C_VEL
LIN {X 0,Y 319.985,Z 187.627,A -85,B 0,C 180,E1 -15302.518,E2 -15302.518} C_VEL
LIN {X 0,Y 319.878,Z 187.638,A -85,B 0,C 180,E1 -15306.537,E2 -15306.537} C_VEL
LIN {X 0,Y 319.733,Z 187.658,A -85,B 0,C 180,E1 -15310.128,E2 -15310.128} C_VEL
LIN {X 0,Y 319.73,Z 187.658,A -85,B 0,C 180,E1 -15313.992,E2 -15313.992} C_VEL
LIN {X 0,Y 319.657,Z 187.669,A -85,B 0,C 180,E1 -15317.927,E2 -15317.927} C_VEL
LIN {X 0,Y 319.613,Z 187.67,A -85,B 0,C 180,E1 -15320.599,E2 -15320.599} C_VEL
LIN {X 0,Y 319.569,Z 187.677,A -85,B 0,C 180,E1 -15323.32,E2 -15323.32} C_VEL
LIN {X 0,Y 319.632,Z 187.67,A -85,B 0,C 180,E1 -15326.088,E2 -15326.088} C_VEL
LIN {X 0,Y 319.587,Z 187.674,A -85,B 0,C 180,E1 -15328.934,E2 -15328.934} C_VEL
LIN {X 0,Y 319.531,Z 187.683,A -85,B 0,C 180,E1 -15331.862,E2 -15331.862} C_VEL
LIN {X 0,Y 319.578,Z 187.679,A -85,B 0,C 180,E1 -15335.543,E2 -15335.543} C_VEL
LIN {X 0,Y 319.557,Z 187.679,A -85,B 0,C 180,E1 -15339.669,E2 -15339.669} C_VEL
LIN {X 0,Y 319.521,Z 187.684,A -85,B 0,C 180,E1 -15343.461,E2 -15343.461} C_VEL
LIN {X 0,Y 319.553,Z 187.682,A -85,B 0,C 180,E1 -15347.017,E2 -15347.017} C_VEL
LIN {X 0,Y 319.544,Z 187.683,A -85,B 0,C 180,E1 -15350.371,E2 -15350.371} C_VEL
LIN {X 0,Y 319.535,Z 187.92,A -85,B 0,C 180,E1 -15352.354,E2 -15352.354} C_VEL
LIN {X 0,Y 319.582,Z 190.558,A -85,B 0,C 180,E1 -15355.127,E2 -15355.127} C_VEL
LIN {X 0,Y 319.425,Z 193.554,A -85,B 0,C 180,E1 -15358.127,E2 -15358.127} C_VEL
LIN {X 0,Y 319.208,Z 197.298,A -85,B 0,C 180,E1 -15361.725,E2 -15361.725} C_VEL
LIN {X 0,Y 318.888,Z 201.139,A -85,B 0,C 180,E1 -15365.245,E2 -15365.245} C_VEL
LIN {X 0,Y 318.791,Z 203.314,A -85,B 0,C 180,E1 -15367.192,E2 -15367.192} C_VEL
LIN {X 0,Y 322.704,Z 217.4,A -85,B 0,C 180,E1 -15368.114,E2 -15368.114} C_VEL
LIN {X 0,Y 325.486,Z 230.018,A -85,B 0,C 180,E1 -15369.144,E2 -15369.144} C_VEL
LIN {X 0,Y 326.853,Z 239.331,A -85,B 0,C 180,E1 -15370.042,E2 -15370.042} C_VEL
LIN {X 0,Y 325.69,Z 250.078,A -85,B 0,C 180,E1 -15371.115,E2 -15371.115} C_VEL
LIN {X 0,Y 324.439,Z 260.242,A -85,B 0,C 180,E1 -15372.389,E2 -15372.389} C_VEL
LIN {X 0,Y 323.229,Z 269.918,A -85,B 0,C 180,E1 -15373.906,E2 -15373.906} C_VEL
LIN {X 0,Y 321.764,Z 279.556,A -85,B 0,C 180,E1 -15375.776,E2 -15375.776} C_VEL
LIN {X 0,Y 320.55,Z 287.241,A -85,B 0,C 180,E1 -15377.657,E2 -15377.657} C_VEL
LIN {X 0,Y 319.439,Z 294.294,A -85,B 0,C 180,E1 -15379.863,E2 -15379.863} C_VEL
LIN {X 0,Y 318.8,Z 298.988,A -85,B 0,C 180,E1 -15381.762,E2 -15381.762} C_VEL
LIN {X 0,Y 318.384,Z 302.578,A -85,B 0,C 180,E1 -15383.664,E2 -15383.664} C_VEL
LIN {X 0,Y 318.193,Z 304.433,A -85,B 0,C 180,E1 -15384.932,E2 -15384.932} C_VEL
LIN {X 0,Y 318.01,Z 305.83,A -85,B 0,C 180,E1 -15386.199,E2 -15386.199} C_VEL
LIN {X 0,Y 317.801,Z 307.434,A -85,B 0,C 180,E1 -15388.733,E2 -15388.733} C_VEL
LIN {X 0,Y 317.791,Z 307.665,A -85,B 0,C 180,E1 -15390,E2 -15390} C_VEL
LIN {X 0,Y 317.801,Z 307.474,A -85,B 0,C 180,E1 -15391.267,E2 -15391.267} C_VEL
LIN {X 0,Y 318.007,Z 305.921,A -85,B 0,C 180,E1 -15393.802,E2 -15393.802} C_VEL
LIN {X 0,Y 318.171,Z 304.564,A -85,B 0,C 180,E1 -15395.069,E2 -15395.069} C_VEL
LIN {X 0,Y 318.469,Z 302.067,A -85,B 0,C 180,E1 -15396.749,E2 -15396.749} C_VEL
LIN {X 0,Y 318.951,Z 297.814,A -85,B 0,C 180,E1 -15398.873,E2 -15398.873} C_VEL
LIN {X 0,Y 319.711,Z 292.798,A -85,B 0,C 180,E1 -15400.769,E2 -15400.769} C_VEL
LIN {X 0,Y 320.707,Z 286.481,A -85,B 0,C 180,E1 -15402.659,E2 -15402.659} C_VEL
LIN {X 0,Y 321.887,Z 278.575,A -85,B 0,C 180,E1 -15404.542,E2 -15404.542} C_VEL
LIN {X 0,Y 323.474,Z 268.734,A -85,B 0,C 180,E1 -15406.407,E2 -15406.407} C_VEL
LIN {X 0,Y 324.686,Z 258.41,A -85,B 0,C 180,E1 -15407.966,E2 -15407.966} C_VEL
LIN {X 0,Y 325.947,Z 248.177,A -85,B 0,C 180,E1 -15409.197,E2 -15409.197} C_VEL
LIN {X 0,Y 326.886,Z 238.741,A -85,B 0,C 180,E1 -15410.121,E2 -15410.121} C_VEL
LIN {X 0,Y 325.023,Z 227.512,A -85,B 0,C 180,E1 -15411.184,E2 -15411.184} C_VEL
LIN {X 0,Y 322.052,Z 214.83,A -85,B 0,C 180,E1 -15412.187,E2 -15412.187} C_VEL
LIN {X 0,Y 318.764,Z 203.301,A -85,B 0,C 180,E1 -15412.937,E2 -15412.937} C_VEL
LIN {X 0,Y 318.968,Z 199.724,A -85,B 0,C 180,E1 -15416.147,E2 -15416.147} C_VEL
LIN {X 0,Y 319.212,Z 196.706,A -85,B 0,C 180,E1 -15418.971,E2 -15418.971} C_VEL
LIN {X 0,Y 319.429,Z 193.689,A -85,B 0,C 180,E1 -15421.873,E2 -15421.873} C_VEL
LIN {X 0,Y 319.639,Z 190.006,A -85,B 0,C 180,E1 -15425.557,E2 -15425.557} C_VEL
LIN {X 0,Y 319.512,Z 187.697,A -85,B 0,C 180,E1 -15428.017,E2 -15428.017} C_VEL
LIN {X 0,Y 319.506,Z 187.685,A -85,B 0,C 180,E1 -15431.593,E2 -15431.593} C_VEL
LIN {X 0,Y 319.489,Z 187.687,A -85,B 0,C 180,E1 -15434.743,E2 -15434.743} C_VEL
LIN {X 0,Y 319.526,Z 187.682,A -85,B 0,C 180,E1 -15438.403,E2 -15438.403} C_VEL
LIN {X 0,Y 319.536,Z 187.68,A -85,B 0,C 180,E1 -15441.987,E2 -15441.987} C_VEL
LIN {X 0,Y 319.561,Z 187.678,A -85,B 0,C 180,E1 -15445.123,E2 -15445.123} C_VEL
LIN {X 0,Y 319.568,Z 187.677,A -85,B 0,C 180,E1 -15449.059,E2 -15449.059} C_VEL
LIN {X 0,Y 319.607,Z 187.675,A -85,B 0,C 180,E1 -15452.498,E2 -15452.498} C_VEL
LIN {X 0,Y 319.634,Z 187.67,A -85,B 0,C 180,E1 -15454.07,E2 -15454.07} C_VEL
LIN {X 0,Y 318.96,Z 187.756,A -85,B 0,C 180,E1 -15455.122,E2 -15455.122} C_VEL
LIN {X 0,Y 316.076,Z 188.113,A -85,B 0,C 180,E1 -15456.833,E2 -15456.833} C_VEL
LIN {X 0,Y 313.646,Z 188.417,A -85,B 0,C 180,E1 -15458.221,E2 -15458.221} C_VEL
LIN {X 0,Y 312.624,Z 188.541,A -85,B 0,C 180,E1 -15459.296,E2 -15459.296} C_VEL
LIN {X 0,Y 312.552,Z 188.548,A -85,B 0,C 180,E1 -15459.66,E2 -15459.66} C_VEL
LIN {X 0,Y 312.608,Z 188.542,A -85,B 0,C 180,E1 -15463.006,E2 -15463.006} C_VEL
LIN {X 0,Y 312.695,Z 188.536,A -85,B 0,C 180,E1 -15465.686,E2 -15465.686} C_VEL
LIN {X 0,Y 312.686,Z 188.538,A -85,B 0,C 180,E1 -15469.641,E2 -15469.641} C_VEL
LIN {X 0,Y 312.797,Z 188.519,A -85,B 0,C 180,E1 -15472.252,E2 -15472.252} C_VEL
LIN {X 0,Y 312.7,Z 188.532,A -85,B 0,C 180,E1 -15474.842,E2 -15474.842} C_VEL
LIN {X 0,Y 312.991,Z 188.496,A -85,B 0,C 180,E1 -15478.713,E2 -15478.713} C_VEL
LIN {X 0,Y 312.991,Z 188.499,A -85,B 0,C 180,E1 -15481.287,E2 -15481.287} C_VEL
LIN {X 0,Y 312.701,Z 188.535,A -85,B 0,C 180,E1 -15485.158,E2 -15485.158} C_VEL
LIN {X 0,Y 312.797,Z 188.52,A -85,B 0,C 180,E1 -15487.748,E2 -15487.748} C_VEL
LIN {X 0,Y 312.672,Z 188.535,A -85,B 0,C 180,E1 -15491.671,E2 -15491.671} C_VEL
LIN {X 0,Y 312.701,Z 188.534,A -85,B 0,C 180,E1 -15494.888,E2 -15494.888} C_VEL
LIN {X 0,Y 312.61,Z 188.543,A -85,B 0,C 180,E1 -15499.225,E2 -15499.225} C_VEL
LIN {X 0,Y 312.527,Z 188.554,A -85,B 0,C 180,E1 -15502.78,E2 -15502.78} C_VEL
LIN {X 0,Y 312.603,Z 188.548,A -85,B 0,C 180,E1 -15505.935,E2 -15505.935} C_VEL
LIN {X 0,Y 312.539,Z 188.555,A -85,B 0,C 180,E1 -15509.651,E2 -15509.651} C_VEL
LIN {X 0,Y 312.52,Z 188.559,A -85,B 0,C 180,E1 -15513.689,E2 -15513.689} C_VEL
LIN {X 0,Y 312.516,Z 188.559,A -85,B 0,C 180,E1 -15517.387,E2 -15517.387} C_VEL
LIN {X 0,Y 312.49,Z 188.56,A -85,B 0,C 180,E1 -15520.709,E2 -15520.709} C_VEL
LIN {X 0,Y 312.516,Z 188.712,A -85,B 0,C 180,E1 -15523.86,E2 -15523.86} C_VEL
LIN {X 0,Y 313.324,Z 193.232,A -85,B 0,C 180,E1 -15527.749,E2 -15527.749} C_VEL
LIN {X 0,Y 313.996,Z 197.515,A -85,B 0,C 180,E1 -15531.192,E2 -15531.192} C_VEL
LIN {X 0,Y 314.224,Z 200.776,A -85,B 0,C 180,E1 -15533.628,E2 -15533.628} C_VEL
LIN {X 0,Y 314.045,Z 204.075,A -85,B 0,C 180,E1 -15535.98,E2 -15535.98} C_VEL
LIN {X 0,Y 313.472,Z 208.374,A -85,B 0,C 180,E1 -15538.958,E2 -15538.958} C_VEL
LIN {X 0,Y 312.788,Z 213.738,A -85,B 0,C 180,E1 -15542.573,E2 -15542.573} C_VEL
LIN {X 0,Y 312.165,Z 219.737,A -85,B 0,C 180,E1 -15546.578,E2 -15546.578} C_VEL
LIN {X 0,Y 315.386,Z 234,A -85,B 0,C 180,E1 -15547.45,E2 -15547.45} C_VEL
LIN {X 0,Y 317.448,Z 246.477,A -85,B 0,C 180,E1 -15548.41,E2 -15548.41} C_VEL
LIN {X 0,Y 318.695,Z 258.162,A -85,B 0,C 180,E1 -15549.507,E2 -15549.507} C_VEL
LIN {X 0,Y 318.858,Z 264.577,A -85,B 0,C 180,E1 -15550.191,E2 -15550.191} C_VEL
LIN {X 0,Y 317.196,Z 276.368,A -85,B 0,C 180,E1 -15551.595,E2 -15551.595} C_VEL
LIN {X 0,Y 315.699,Z 286.845,A -85,B 0,C 180,E1 -15553.178,E2 -15553.178} C_VEL
LIN {X 0,Y 314.469,Z 295.328,A -85,B 0,C 180,E1 -15554.775,E2 -15554.775} C_VEL
LIN {X 0,Y 313.195,Z 303.607,A -85,B 0,C 180,E1 -15556.702,E2 -15556.702} C_VEL
LIN {X 0,Y 312.221,Z 310.284,A -85,B 0,C 180,E1 -15558.64,E2 -15558.64} C_VEL
LIN {X 0,Y 311.422,Z 316.395,A -85,B 0,C 180,E1 -15560.911,E2 -15560.911} C_VEL
LIN {X 0,Y 311,Z 320.369,A -85,B 0,C 180,E1 -15562.86,E2 -15562.86} C_VEL
LIN {X 0,Y 310.763,Z 323.307,A -85,B 0,C 180,E1 -15564.81,E2 -15564.81} C_VEL
LIN {X 0,Y 310.731,Z 324.706,A -85,B 0,C 180,E1 -15566.109,E2 -15566.109} C_VEL
LIN {X 0,Y 310.683,Z 325.704,A -85,B 0,C 180,E1 -15567.407,E2 -15567.407} C_VEL
LIN {X 0,Y 310.642,Z 326.313,A -85,B 0,C 180,E1 -15568.703,E2 -15568.703} C_VEL
LIN {X 0,Y 310.656,Z 326.529,A -85,B 0,C 180,E1 -15570,E2 -15570} C_VEL
LIN {X 0,Y 310.642,Z 326.31,A -85,B 0,C 180,E1 -15571.296,E2 -15571.296} C_VEL
LIN {X 0,Y 310.683,Z 325.7,A -85,B 0,C 180,E1 -15572.593,E2 -15572.593} C_VEL
LIN {X 0,Y 310.732,Z 324.7,A -85,B 0,C 180,E1 -15573.89,E2 -15573.89} C_VEL
LIN {X 0,Y 310.813,Z 322.484,A -85,B 0,C 180,E1 -15575.781,E2 -15575.781} C_VEL
LIN {X 0,Y 311.079,Z 319.121,A -85,B 0,C 180,E1 -15577.79,E2 -15577.79} C_VEL
LIN {X 0,Y 311.619,Z 314.773,A -85,B 0,C 180,E1 -15579.738,E2 -15579.738} C_VEL
LIN {X 0,Y 312.322,Z 309.234,A -85,B 0,C 180,E1 -15581.684,E2 -15581.684} C_VEL
LIN {X 0,Y 313.401,Z 302.327,A -85,B 0,C 180,E1 -15583.618,E2 -15583.618} C_VEL
LIN {X 0,Y 314.457,Z 295.275,A -85,B 0,C 180,E1 -15585.224,E2 -15585.224} C_VEL
LIN {X 0,Y 315.713,Z 286.778,A -85,B 0,C 180,E1 -15586.821,E2 -15586.821} C_VEL
LIN {X 0,Y 317.145,Z 276.279,A -85,B 0,C 180,E1 -15588.408,E2 -15588.408} C_VEL
LIN {X 0,Y 318.784,Z 264.469,A -85,B 0,C 180,E1 -15589.813,E2 -15589.813} C_VEL
LIN {X 0,Y 318.695,Z 258.028,A -85,B 0,C 180,E1 -15590.492,E2 -15590.492} C_VEL
LIN {X 0,Y 317.435,Z 246.372,A -85,B 0,C 180,E1 -15591.584,E2 -15591.584} C_VEL
LIN {X 0,Y 315.162,Z 232.972,A -85,B 0,C 180,E1 -15592.609,E2 -15592.609} C_VEL
LIN {X 0,Y 312.172,Z 219.718,A -85,B 0,C 180,E1 -15593.42,E2 -15593.42} C_VEL
LIN {X 0,Y 312.786,Z 213.716,A -85,B 0,C 180,E1 -15597.426,E2 -15597.426} C_VEL
LIN {X 0,Y 313.468,Z 208.358,A -85,B 0,C 180,E1 -15601.041,E2 -15601.041} C_VEL
LIN {X 0,Y 314.073,Z 203.914,A -85,B 0,C 180,E1 -15604.111,E2 -15604.111} C_VEL
LIN {X 0,Y 314.211,Z 199.683,A -85,B 0,C 180,E1 -15607.15,E2 -15607.15} C_VEL
LIN {X 0,Y 313.732,Z 195.494,A -85,B 0,C 180,E1 -15610.391,E2 -15610.391} C_VEL
LIN {X 0,Y 312.911,Z 190.969,A -85,B 0,C 180,E1 -15614.127,E2 -15614.127} C_VEL
LIN {X 0,Y 312.493,Z 188.567,A -85,B 0,C 180,E1 -15616.406,E2 -15616.406} C_VEL
LIN {X 0,Y 312.502,Z 188.559,A -85,B 0,C 180,E1 -15619.874,E2 -15619.874} C_VEL
LIN {X 0,Y 312.532,Z 188.556,A -85,B 0,C 180,E1 -15624.05,E2 -15624.05} C_VEL
LIN {X 0,Y 312.502,Z 188.557,A -85,B 0,C 180,E1 -15627.333,E2 -15627.333} C_VEL
LIN {X 0,Y 312.542,Z 188.551,A -85,B 0,C 180,E1 -15631.279,E2 -15631.279} C_VEL
LIN {X 0,Y 312.583,Z 188.547,A -85,B 0,C 180,E1 -15634.711,E2 -15634.711} C_VEL
LIN {X 0,Y 312.536,Z 188.553,A -85,B 0,C 180,E1 -15638.913,E2 -15638.913} C_VEL
LIN {X 0,Y 312.636,Z 188.544,A -85,B 0,C 180,E1 -15641.656,E2 -15641.656} C_VEL
LIN {X 0,Y 312.692,Z 188.536,A -85,B 0,C 180,E1 -15645.686,E2 -15645.686} C_VEL
LIN {X 0,Y 312.683,Z 188.535,A -85,B 0,C 180,E1 -15649.641,E2 -15649.641} C_VEL
LIN {X 0,Y 312.794,Z 188.52,A -85,B 0,C 180,E1 -15652.252,E2 -15652.252} C_VEL
LIN {X 0,Y 312.698,Z 188.535,A -85,B 0,C 180,E1 -15654.842,E2 -15654.842} C_VEL
LIN {X 0,Y 312.988,Z 188.499,A -85,B 0,C 180,E1 -15658.713,E2 -15658.713} C_VEL
LIN {X 0,Y 312.988,Z 188.497,A -85,B 0,C 180,E1 -15661.287,E2 -15661.287} C_VEL
LIN {X 0,Y 312.698,Z 188.533,A -85,B 0,C 180,E1 -15665.158,E2 -15665.158} C_VEL
LIN {X 0,Y 312.794,Z 188.52,A -85,B 0,C 180,E1 -15667.748,E2 -15667.748} C_VEL
LIN {X 0,Y 312.661,Z 188.537,A -85,B 0,C 180,E1 -15671.672,E2 -15671.672} C_VEL
LIN {X 0,Y 312.698,Z 188.532,A -85,B 0,C 180,E1 -15674.888,E2 -15674.888} C_VEL
LIN {X 0,Y 312.629,Z 188.54,A -85,B 0,C 180,E1 -15679.237,E2 -15679.237} C_VEL
LIN {X 0,Y 312.544,Z 188.551,A -85,B 0,C 180,E1 -15682.79,E2 -15682.79} C_VEL
LIN {X 0,Y 312.601,Z 188.548,A -85,B 0,C 180,E1 -15685.936,E2 -15685.936} C_VEL
LIN {X 0,Y 312.544,Z 188.555,A -85,B 0,C 180,E1 -15689.65,E2 -15689.65} C_VEL
LIN {X 0,Y 312.518,Z 188.557,A -85,B 0,C 180,E1 -15693.689,E2 -15693.689} C_VEL
LIN {X 0,Y 312.514,Z 188.559,A -85,B 0,C 180,E1 -15697.387,E2 -15697.387} C_VEL
LIN {X 0,Y 312.488,Z 188.56,A -85,B 0,C 180,E1 -15700.71,E2 -15700.71} C_VEL
LIN {X 0,Y 312.451,Z 188.563,A -85,B 0,C 180,E1 -15704.21,E2 -15704.21} C_VEL
LIN {X 0,Y 312.484,Z 188.56,A -85,B 0,C 180,E1 -15707.919,E2 -15707.919} C_VEL
LIN {X 0,Y 312.492,Z 188.562,A -85,B 0,C 180,E1 -15710.971,E2 -15710.971} C_VEL
LIN {X 0,Y 312.495,Z 188.628,A -85,B 0,C 180,E1 -15711.92,E2 -15711.92} C_VEL
LIN {X 0,Y 312.58,Z 190.749,A -85,B 0,C 180,E1 -15714.227,E2 -15714.227} C_VEL
LIN {X 0,Y 312.442,Z 193.751,A -85,B 0,C 180,E1 -15717.327,E2 -15717.327} C_VEL
LIN {X 0,Y 312.19,Z 197.879,A -85,B 0,C 180,E1 -15721.398,E2 -15721.398} C_VEL
LIN {X 0,Y 311.907,Z 201.348,A -85,B 0,C 180,E1 -15724.653,E2 -15724.653} C_VEL
LIN {X 0,Y 311.761,Z 203.557,A -85,B 0,C 180,E1 -15726.656,E2 -15726.656} C_VEL
LIN {X 0,Y 315.51,Z 216.617,A -85,B 0,C 180,E1 -15727.53,E2 -15727.53} C_VEL
LIN {X 0,Y 318.317,Z 228.947,A -85,B 0,C 180,E1 -15728.552,E2 -15728.552} C_VEL
LIN {X 0,Y 320.083,Z 239.555,A -85,B 0,C 180,E1 -15729.601,E2 -15729.601} C_VEL
LIN {X 0,Y 318.999,Z 250.295,A -85,B 0,C 180,E1 -15730.703,E2 -15730.703} C_VEL
LIN {X 0,Y 317.605,Z 261.021,A -85,B 0,C 180,E1 -15732.085,E2 -15732.085} C_VEL
LIN {X 0,Y 316.427,Z 270.134,A -85,B 0,C 180,E1 -15733.55,E2 -15733.55} C_VEL
LIN {X 0,Y 314.89,Z 279.772,A -85,B 0,C 180,E1 -15735.458,E2 -15735.458} C_VEL
LIN {X 0,Y 313.619,Z 287.456,A -85,B 0,C 180,E1 -15737.38,E2 -15737.38} C_VEL
LIN {X 0,Y 312.461,Z 294.508,A -85,B 0,C 180,E1 -15739.634,E2 -15739.634} C_VEL
LIN {X 0,Y 311.781,Z 299.202,A -85,B 0,C 180,E1 -15741.575,E2 -15741.575} C_VEL
LIN {X 0,Y 311.332,Z 302.792,A -85,B 0,C 180,E1 -15743.52,E2 -15743.52} C_VEL
LIN {X 0,Y 311.125,Z 304.647,A -85,B 0,C 180,E1 -15744.816,E2 -15744.816} C_VEL
LIN {X 0,Y 310.947,Z 306.043,A -85,B 0,C 180,E1 -15746.112,E2 -15746.112} C_VEL
LIN {X 0,Y 310.714,Z 307.647,A -85,B 0,C 180,E1 -15748.704,E2 -15748.704} C_VEL
LIN {X 0,Y 310.701,Z 307.878,A -85,B 0,C 180,E1 -15750,E2 -15750} C_VEL
LIN {X 0,Y 310.714,Z 307.687,A -85,B 0,C 180,E1 -15751.296,E2 -15751.296} C_VEL
LIN {X 0,Y 310.943,Z 306.133,A -85,B 0,C 180,E1 -15753.888,E2 -15753.888} C_VEL
LIN {X 0,Y 311.105,Z 304.776,A -85,B 0,C 180,E1 -15755.185,E2 -15755.185} C_VEL
LIN {X 0,Y 311.363,Z 302.602,A -85,B 0,C 180,E1 -15756.705,E2 -15756.705} C_VEL
LIN {X 0,Y 311.942,Z 298.026,A -85,B 0,C 180,E1 -15759.074,E2 -15759.074} C_VEL
LIN {X 0,Y 312.73,Z 293.01,A -85,B 0,C 180,E1 -15761.013,E2 -15761.013} C_VEL
LIN {X 0,Y 313.791,Z 286.691,A -85,B 0,C 180,E1 -15762.943,E2 -15762.943} C_VEL
LIN {X 0,Y 315.026,Z 278.785,A -85,B 0,C 180,E1 -15764.866,E2 -15764.866} C_VEL
LIN {X 0,Y 316.385,Z 270.719,A -85,B 0,C 180,E1 -15766.453,E2 -15766.453} C_VEL
LIN {X 0,Y 317.675,Z 260.883,A -85,B 0,C 180,E1 -15768.043,E2 -15768.043} C_VEL
LIN {X 0,Y 319.064,Z 249.808,A -85,B 0,C 180,E1 -15769.461,E2 -15769.461} C_VEL
LIN {X 0,Y 320.173,Z 240.704,A -85,B 0,C 180,E1 -15770.394,E2 -15770.394} C_VEL
LIN {X 0,Y 318.401,Z 229.203,A -85,B 0,C 180,E1 -15771.534,E2 -15771.534} C_VEL
LIN {X 0,Y 315.594,Z 216.937,A -85,B 0,C 180,E1 -15772.558,E2 -15772.558} C_VEL
LIN {X 0,Y 311.742,Z 203.536,A -85,B 0,C 180,E1 -15773.475,E2 -15773.475} C_VEL
LIN {X 0,Y 311.968,Z 199.932,A -85,B 0,C 180,E1 -15776.78,E2 -15776.78} C_VEL
LIN {X 0,Y 312.225,Z 196.914,A -85,B 0,C 180,E1 -15779.684,E2 -15779.684} C_VEL
LIN {X 0,Y 312.526,Z 192.872,A -85,B 0,C 180,E1 -15783.69,E2 -15783.69} C_VEL
LIN {X 0,Y 312.611,Z 190.672,A -85,B 0,C 180,E1 -15785.968,E2 -15785.968} C_VEL
LIN {X 0,Y 312.502,Z 188.732,A -85,B 0,C 180,E1 -15788.081,E2 -15788.081} C_VEL
LIN {X 0,Y 312.456,Z 188.561,A -85,B 0,C 180,E1 -15792.075,E2 -15792.075} C_VEL
LIN {X 0,Y 312.459,Z 188.561,A -85,B 0,C 180,E1 -15796.035,E2 -15796.035} C_VEL
LIN {X 0,Y 312.505,Z 188.556,A -85,B 0,C 180,E1 -15799.875,E2 -15799.875} C_VEL
LIN {X 0,Y 312.535,Z 188.553,A -85,B 0,C 180,E1 -15804.051,E2 -15804.051} C_VEL
LIN {X 0,Y 312.505,Z 188.555,A -85,B 0,C 180,E1 -15807.334,E2 -15807.334} C_VEL
LIN {X 0,Y 312.546,Z 188.55,A -85,B 0,C 180,E1 -15811.279,E2 -15811.279} C_VEL
LIN {X 0,Y 312.587,Z 188.547,A -85,B 0,C 180,E1 -15814.711,E2 -15814.711} C_VEL
LIN {X 0,Y 312.589,Z 188.545,A -85,B 0,C 180,E1 -15817.529,E2 -15817.529} C_VEL
LIN {X 0,Y 312.552,Z 188.548,A -85,B 0,C 180,E1 -15819.66,E2 -15819.66} C_VEL
LIN {X 0,Y 311.945,Z 188.628,A -85,B 0,C 180,E1 -15820.735,E2 -15820.735} C_VEL
LIN {X 0,Y 309.209,Z 188.975,A -85,B 0,C 180,E1 -15822.488,E2 -15822.488} C_VEL
LIN {X 0,Y 306.834,Z 189.271,A -85,B 0,C 180,E1 -15823.908,E2 -15823.908} C_VEL
LIN {X 0,Y 305.762,Z 189.4,A -85,B 0,C 180,E1 -15825.006,E2 -15825.006} C_VEL
LIN {X 0,Y 305.647,Z 189.411,A -85,B 0,C 180,E1 -15825.378,E2 -15825.378} C_VEL
LIN {X 0,Y 305.625,Z 189.416,A -85,B 0,C 180,E1 -15829.399,E2 -15829.399} C_VEL
LIN {X 0,Y 305.747,Z 189.398,A -85,B 0,C 180,E1 -15832.073,E2 -15832.073} C_VEL
LIN {X 0,Y 305.668,Z 189.408,A -85,B 0,C 180,E1 -15834.723,E2 -15834.723} C_VEL
LIN {X 0,Y 305.958,Z 189.372,A -85,B 0,C 180,E1 -15838.684,E2 -15838.684} C_VEL
LIN {X 0,Y 305.958,Z 189.375,A -85,B 0,C 180,E1 -15841.316,E2 -15841.316} C_VEL
LIN {X 0,Y 305.67,Z 189.41,A -85,B 0,C 180,E1 -15845.277,E2 -15845.277} C_VEL
LIN {X 0,Y 305.747,Z 189.398,A -85,B 0,C 180,E1 -15847.927,E2 -15847.927} C_VEL
LIN {X 0,Y 305.607,Z 189.416,A -85,B 0,C 180,E1 -15851.945,E2 -15851.945} C_VEL
LIN {X 0,Y 305.639,Z 189.413,A -85,B 0,C 180,E1 -15855.035,E2 -15855.035} C_VEL
LIN {X 0,Y 305.581,Z 189.421,A -85,B 0,C 180,E1 -15858.783,E2 -15858.783} C_VEL
LIN {X 0,Y 305.487,Z 189.43,A -85,B 0,C 180,E1 -15863.039,E2 -15863.039} C_VEL
LIN {X 0,Y 305.548,Z 189.427,A -85,B 0,C 180,E1 -15866.227,E2 -15866.227} C_VEL
LIN {X 0,Y 305.489,Z 189.431,A -85,B 0,C 180,E1 -15869.047,E2 -15869.047} C_VEL
LIN {X 0,Y 305.444,Z 189.441,A -85,B 0,C 180,E1 -15871.952,E2 -15871.952} C_VEL
LIN {X 0,Y 305.463,Z 189.436,A -85,B 0,C 180,E1 -15875.113,E2 -15875.113} C_VEL
LIN {X 0,Y 305.436,Z 189.438,A -85,B 0,C 180,E1 -15878.525,E2 -15878.525} C_VEL
LIN {X 0,Y 305.463,Z 189.437,A -85,B 0,C 180,E1 -15882.587,E2 -15882.587} C_VEL
LIN {X 0,Y 305.468,Z 189.531,A -85,B 0,C 180,E1 -15883.352,E2 -15883.352} C_VEL
LIN {X 0,Y 306.24,Z 193.908,A -85,B 0,C 180,E1 -15887.255,E2 -15887.255} C_VEL
LIN {X 0,Y 306.791,Z 197.364,A -85,B 0,C 180,E1 -15890.101,E2 -15890.101} C_VEL
LIN {X 0,Y 307.192,Z 201.306,A -85,B 0,C 180,E1 -15893.201,E2 -15893.201} C_VEL
LIN {X 0,Y 307.097,Z 204.394,A -85,B 0,C 180,E1 -15895.474,E2 -15895.474} C_VEL
LIN {X 0,Y 306.442,Z 209.247,A -85,B 0,C 180,E1 -15898.934,E2 -15898.934} C_VEL
LIN {X 0,Y 305.733,Z 214.599,A -85,B 0,C 180,E1 -15902.629,E2 -15902.629} C_VEL
LIN {X 0,Y 305.167,Z 219.532,A -85,B 0,C 180,E1 -15906.004,E2 -15906.004} C_VEL
LIN {X 0,Y 308.572,Z 234.358,A -85,B 0,C 180,E1 -15906.957,E2 -15906.957} C_VEL
LIN {X 0,Y 310.732,Z 247.585,A -85,B 0,C 180,E1 -15908.021,E2 -15908.021} C_VEL
LIN {X 0,Y 311.958,Z 259.64,A -85,B 0,C 180,E1 -15909.217,E2 -15909.217} C_VEL
LIN {X 0,Y 312.143,Z 264.367,A -85,B 0,C 180,E1 -15909.746,E2 -15909.746} C_VEL
LIN {X 0,Y 310.457,Z 276.159,A -85,B 0,C 180,E1 -15911.18,E2 -15911.18} C_VEL
LIN {X 0,Y 309.168,Z 284.686,A -85,B 0,C 180,E1 -15912.47,E2 -15912.47} C_VEL
LIN {X 0,Y 307.846,Z 293.532,A -85,B 0,C 180,E1 -15914.1,E2 -15914.1} C_VEL
LIN {X 0,Y 306.69,Z 300.837,A -85,B 0,C 180,E1 -15915.739,E2 -15915.739} C_VEL
LIN {X 0,Y 305.494,Z 308.031,A -85,B 0,C 180,E1 -15917.713,E2 -15917.713} C_VEL
LIN {X 0,Y 304.804,Z 312.891,A -85,B 0,C 180,E1 -15919.37,E2 -15919.37} C_VEL
LIN {X 0,Y 304.195,Z 317.617,A -85,B 0,C 180,E1 -15921.363,E2 -15921.363} C_VEL
LIN {X 0,Y 303.837,Z 321.23,A -85,B 0,C 180,E1 -15923.358,E2 -15923.358} C_VEL
LIN {X 0,Y 303.686,Z 323.094,A -85,B 0,C 180,E1 -15924.688,E2 -15924.688} C_VEL
LIN {X 0,Y 303.647,Z 324.494,A -85,B 0,C 180,E1 -15926.018,E2 -15926.018} C_VEL
LIN {X 0,Y 303.608,Z 325.492,A -85,B 0,C 180,E1 -15927.346,E2 -15927.346} C_VEL
LIN {X 0,Y 303.56,Z 326.101,A -85,B 0,C 180,E1 -15928.673,E2 -15928.673} C_VEL
LIN {X 0,Y 303.57,Z 326.316,A -85,B 0,C 180,E1 -15930,E2 -15930} C_VEL
LIN {X 0,Y 303.56,Z 326.097,A -85,B 0,C 180,E1 -15931.326,E2 -15931.326} C_VEL
LIN {X 0,Y 303.608,Z 325.487,A -85,B 0,C 180,E1 -15932.653,E2 -15932.653} C_VEL
LIN {X 0,Y 303.647,Z 324.487,A -85,B 0,C 180,E1 -15933.981,E2 -15933.981} C_VEL
LIN {X 0,Y 303.73,Z 322.504,A -85,B 0,C 180,E1 -15935.744,E2 -15935.744} C_VEL
LIN {X 0,Y 304.033,Z 318.906,A -85,B 0,C 180,E1 -15937.972,E2 -15937.972} C_VEL
LIN {X 0,Y 304.579,Z 314.557,A -85,B 0,C 180,E1 -15939.965,E2 -15939.965} C_VEL
LIN {X 0,Y 305.322,Z 309.018,A -85,B 0,C 180,E1 -15941.956,E2 -15941.956} C_VEL
LIN {X 0,Y 306.457,Z 302.111,A -85,B 0,C 180,E1 -15943.933,E2 -15943.933} C_VEL
LIN {X 0,Y 307.577,Z 295.058,A -85,B 0,C 180,E1 -15945.574,E2 -15945.574} C_VEL
LIN {X 0,Y 308.902,Z 286.561,A -85,B 0,C 180,E1 -15947.203,E2 -15947.203} C_VEL
LIN {X 0,Y 310.38,Z 276.061,A -85,B 0,C 180,E1 -15948.824,E2 -15948.824} C_VEL
LIN {X 0,Y 312.089,Z 264.251,A -85,B 0,C 180,E1 -15950.257,E2 -15950.257} C_VEL
LIN {X 0,Y 311.529,Z 254.768,A -85,B 0,C 180,E1 -15951.28,E2 -15951.28} C_VEL
LIN {X 0,Y 310.001,Z 242.841,A -85,B 0,C 180,E1 -15952.378,E2 -15952.378} C_VEL
LIN {X 0,Y 307.776,Z 230.654,A -85,B 0,C 180,E1 -15953.288,E2 -15953.288} C_VEL
LIN {X 0,Y 305.178,Z 219.557,A -85,B 0,C 180,E1 -15953.961,E2 -15953.961} C_VEL
LIN {X 0,Y 305.859,Z 213.511,A -85,B 0,C 180,E1 -15958.102,E2 -15958.102} C_VEL
LIN {X 0,Y 306.609,Z 207.915,A -85,B 0,C 180,E1 -15961.994,E2 -15961.994} C_VEL
LIN {X 0,Y 307.157,Z 203.861,A -85,B 0,C 180,E1 -15964.891,E2 -15964.891} C_VEL
LIN {X 0,Y 307.196,Z 201.274,A -85,B 0,C 180,E1 -15966.8,E2 -15966.8} C_VEL
LIN {X 0,Y 306.807,Z 197.351,A -85,B 0,C 180,E1 -15969.895,E2 -15969.895} C_VEL
LIN {X 0,Y 306.084,Z 192.969,A -85,B 0,C 180,E1 -15973.537,E2 -15973.537} C_VEL
LIN {X 0,Y 305.47,Z 189.439,A -85,B 0,C 180,E1 -15976.796,E2 -15976.796} C_VEL
LIN {X 0,Y 305.456,Z 189.437,A -85,B 0,C 180,E1 -15979.892,E2 -15979.892} C_VEL
LIN {X 0,Y 305.461,Z 189.435,A -85,B 0,C 180,E1 -15983.636,E2 -15983.636} C_VEL
LIN {X 0,Y 305.463,Z 189.437,A -85,B 0,C 180,E1 -15986.483,E2 -15986.483} C_VEL
LIN {X 0,Y 305.456,Z 189.435,A -85,B 0,C 180,E1 -15989.59,E2 -15989.59} C_VEL
LIN {X 0,Y 305.516,Z 189.428,A -85,B 0,C 180,E1 -15992.608,E2 -15992.608} C_VEL
LIN {X 0,Y 305.503,Z 189.431,A -85,B 0,C 180,E1 -15995.538,E2 -15995.538} C_VEL
LIN {X 0,Y 305.51,Z 189.432,A -85,B 0,C 180,E1 -15999.814,E2 -15999.814} C_VEL
LIN {X 0,Y 305.572,Z 189.42,A -85,B 0,C 180,E1 -16002.603,E2 -16002.603} C_VEL
LIN {X 0,Y 305.647,Z 189.414,A -85,B 0,C 180,E1 -16005.349,E2 -16005.349} C_VEL
LIN {X 0,Y 305.622,Z 189.415,A -85,B 0,C 180,E1 -16009.399,E2 -16009.399} C_VEL
LIN {X 0,Y 305.744,Z 189.398,A -85,B 0,C 180,E1 -16012.073,E2 -16012.073} C_VEL
LIN {X 0,Y 305.667,Z 189.41,A -85,B 0,C 180,E1 -16014.723,E2 -16014.723} C_VEL
LIN {X 0,Y 305.955,Z 189.374,A -85,B 0,C 180,E1 -16018.684,E2 -16018.684} C_VEL
LIN {X 0,Y 305.955,Z 189.373,A -85,B 0,C 180,E1 -16021.316,E2 -16021.316} C_VEL
LIN {X 0,Y 305.667,Z 189.408,A -85,B 0,C 180,E1 -16025.277,E2 -16025.277} C_VEL
LIN {X 0,Y 305.744,Z 189.398,A -85,B 0,C 180,E1 -16027.928,E2 -16027.928} C_VEL
LIN {X 0,Y 305.597,Z 189.418,A -85,B 0,C 180,E1 -16031.945,E2 -16031.945} C_VEL
LIN {X 0,Y 305.636,Z 189.411,A -85,B 0,C 180,E1 -16035.035,E2 -16035.035} C_VEL
LIN {X 0,Y 305.575,Z 189.42,A -85,B 0,C 180,E1 -16039.445,E2 -16039.445} C_VEL
LIN {X 0,Y 305.489,Z 189.43,A -85,B 0,C 180,E1 -16043.042,E2 -16043.042} C_VEL
LIN {X 0,Y 305.53,Z 189.426,A -85,B 0,C 180,E1 -16046.221,E2 -16046.221} C_VEL
LIN {X 0,Y 305.493,Z 189.43,A -85,B 0,C 180,E1 -16049.05,E2 -16049.05} C_VEL
LIN {X 0,Y 305.443,Z 189.437,A -85,B 0,C 180,E1 -16051.952,E2 -16051.952} C_VEL
LIN {X 0,Y 305.46,Z 189.437,A -85,B 0,C 180,E1 -16055.114,E2 -16055.114} C_VEL
LIN {X 0,Y 305.433,Z 189.438,A -85,B 0,C 180,E1 -16058.526,E2 -16058.526} C_VEL
LIN {X 0,Y 305.439,Z 189.437,A -85,B 0,C 180,E1 -16061.857,E2 -16061.857} C_VEL
LIN {X 0,Y 305.399,Z 189.442,A -85,B 0,C 180,E1 -16065.512,E2 -16065.512} C_VEL
LIN {X 0,Y 305.44,Z 189.438,A -85,B 0,C 180,E1 -16068.144,E2 -16068.144} C_VEL
LIN {X 0,Y 305.447,Z 189.452,A -85,B 0,C 180,E1 -16071.594,E2 -16071.594} C_VEL
LIN {X 0,Y 305.507,Z 192.442,A -85,B 0,C 180,E1 -16074.893,E2 -16074.893} C_VEL
LIN {X 0,Y 305.345,Z 195.796,A -85,B 0,C 180,E1 -16078.388,E2 -16078.388} C_VEL
LIN {X 0,Y 305.167,Z 198.493,A -85,B 0,C 180,E1 -16081.078,E2 -16081.078} C_VEL
LIN {X 0,Y 304.767,Z 203.115,A -85,B 0,C 180,E1 -16085.476,E2 -16085.476} C_VEL
LIN {X 0,Y 304.735,Z 203.754,A -85,B 0,C 180,E1 -16086.074,E2 -16086.074} C_VEL
LIN {X 0,Y 308.752,Z 217.538,A -85,B 0,C 180,E1 -16087.051,E2 -16087.051} C_VEL
LIN {X 0,Y 311.354,Z 228.912,A -85,B 0,C 180,E1 -16088.027,E2 -16088.027} C_VEL
LIN {X 0,Y 313.203,Z 239.782,A -85,B 0,C 180,E1 -16089.132,E2 -16089.132} C_VEL
LIN {X 0,Y 313.03,Z 244.667,A -85,B 0,C 180,E1 -16089.635,E2 -16089.635} C_VEL
LIN {X 0,Y 311.617,Z 255.711,A -85,B 0,C 180,E1 -16090.912,E2 -16090.912} C_VEL
LIN {X 0,Y 310.413,Z 265.069,A -85,B 0,C 180,E1 -16092.275,E2 -16092.275} C_VEL
LIN {X 0,Y 309.07,Z 273.815,A -85,B 0,C 180,E1 -16093.826,E2 -16093.826} C_VEL
LIN {X 0,Y 307.486,Z 282.724,A -85,B 0,C 180,E1 -16095.777,E2 -16095.777} C_VEL
LIN {X 0,Y 306.337,Z 289.89,A -85,B 0,C 180,E1 -16097.748,E2 -16097.748} C_VEL
LIN {X 0,Y 305.466,Z 294.723,A -85,B 0,C 180,E1 -16099.394,E2 -16099.394} C_VEL
LIN {X 0,Y 304.742,Z 299.417,A -85,B 0,C 180,E1 -16101.379,E2 -16101.379} C_VEL
LIN {X 0,Y 304.281,Z 303.006,A -85,B 0,C 180,E1 -16103.369,E2 -16103.369} C_VEL
LIN {X 0,Y 304.06,Z 304.86,A -85,B 0,C 180,E1 -16104.695,E2 -16104.695} C_VEL
LIN {X 0,Y 303.886,Z 306.255,A -85,B 0,C 180,E1 -16106.022,E2 -16106.022} C_VEL
LIN {X 0,Y 303.63,Z 307.86,A -85,B 0,C 180,E1 -16108.674,E2 -16108.674} C_VEL
LIN {X 0,Y 303.614,Z 308.091,A -85,B 0,C 180,E1 -16110,E2 -16110} C_VEL
LIN {X 0,Y 303.63,Z 307.899,A -85,B 0,C 180,E1 -16111.327,E2 -16111.327} C_VEL
LIN {X 0,Y 303.881,Z 306.345,A -85,B 0,C 180,E1 -16113.979,E2 -16113.979} C_VEL
LIN {X 0,Y 304.043,Z 304.989,A -85,B 0,C 180,E1 -16115.305,E2 -16115.305} C_VEL
LIN {X 0,Y 304.376,Z 302.229,A -85,B 0,C 180,E1 -16117.23,E2 -16117.23} C_VEL
LIN {X 0,Y 304.923,Z 298.238,A -85,B 0,C 180,E1 -16119.285,E2 -16119.285} C_VEL
LIN {X 0,Y 305.745,Z 293.222,A -85,B 0,C 180,E1 -16121.267,E2 -16121.267} C_VEL
LIN {X 0,Y 306.868,Z 286.902,A -85,B 0,C 180,E1 -16123.24,E2 -16123.24} C_VEL
LIN {X 0,Y 308.181,Z 278.995,A -85,B 0,C 180,E1 -16125.204,E2 -16125.204} C_VEL
LIN {X 0,Y 309.596,Z 270.929,A -85,B 0,C 180,E1 -16126.824,E2 -16126.824} C_VEL
LIN {X 0,Y 310.91,Z 261.093,A -85,B 0,C 180,E1 -16128.45,E2 -16128.45} C_VEL
LIN {X 0,Y 312.38,Z 250.015,A -85,B 0,C 180,E1 -16129.895,E2 -16129.895} C_VEL
LIN {X 0,Y 313.394,Z 240.915,A -85,B 0,C 180,E1 -16130.855,E2 -16130.855} C_VEL
LIN {X 0,Y 311.519,Z 229.547,A -85,B 0,C 180,E1 -16132.025,E2 -16132.025} C_VEL
LIN {X 0,Y 308.831,Z 217.864,A -85,B 0,C 180,E1 -16133.039,E2 -16133.039} C_VEL
LIN {X 0,Y 305.133,Z 205.584,A -85,B 0,C 180,E1 -16133.931,E2 -16133.931} C_VEL
LIN {X 0,Y 304.72,Z 203.737,A -85,B 0,C 180,E1 -16134.062,E2 -16134.062} C_VEL
LIN {X 0,Y 304.981,Z 200.141,A -85,B 0,C 180,E1 -16137.444,E2 -16137.444} C_VEL
LIN {X 0,Y 305.232,Z 197.112,A -85,B 0,C 180,E1 -16140.435,E2 -16140.435} C_VEL
LIN {X 0,Y 305.513,Z 193.523,A -85,B 0,C 180,E1 -16144.091,E2 -16144.091} C_VEL
LIN {X 0,Y 305.55,Z 191.058,A -85,B 0,C 180,E1 -16146.729,E2 -16146.729} C_VEL
LIN {X 0,Y 305.418,Z 189.463,A -85,B 0,C 180,E1 -16148.521,E2 -16148.521} C_VEL
LIN {X 0,Y 305.437,Z 189.436,A -85,B 0,C 180,E1 -16152.582,E2 -16152.582} C_VEL
LIN {X 0,Y 305.427,Z 189.438,A -85,B 0,C 180,E1 -16156.345,E2 -16156.345} C_VEL
LIN {X 0,Y 305.459,Z 189.434,A -85,B 0,C 180,E1 -16159.892,E2 -16159.892} C_VEL
LIN {X 0,Y 305.464,Z 189.433,A -85,B 0,C 180,E1 -16163.636,E2 -16163.636} C_VEL
LIN {X 0,Y 305.467,Z 189.436,A -85,B 0,C 180,E1 -16166.483,E2 -16166.483} C_VEL
LIN {X 0,Y 305.459,Z 189.434,A -85,B 0,C 180,E1 -16169.59,E2 -16169.59} C_VEL
LIN {X 0,Y 305.52,Z 189.428,A -85,B 0,C 180,E1 -16172.608,E2 -16172.608} C_VEL
LIN {X 0,Y 305.509,Z 189.428,A -85,B 0,C 180,E1 -16175.539,E2 -16175.539} C_VEL
LIN {X 0,Y 305.521,Z 189.429,A -85,B 0,C 180,E1 -16179.815,E2 -16179.815} C_VEL
LIN {X 0,Y 305.576,Z 189.418,A -85,B 0,C 180,E1 -16182.603,E2 -16182.603} C_VEL
LIN {X 0,Y 305.647,Z 189.411,A -85,B 0,C 180,E1 -16185.378,E2 -16185.378} C_VEL
LIN {X 0,Y 304.928,Z 189.501,A -85,B 0,C 180,E1 -16186.478,E2 -16186.478} C_VEL
LIN {X 0,Y 302.14,Z 189.848,A -85,B 0,C 180,E1 -16188.271,E2 -16188.271} C_VEL
LIN {X 0,Y 299.809,Z 190.141,A -85,B 0,C 180,E1 -16189.725,E2 -16189.725} C_VEL
LIN {X 0,Y 298.798,Z 190.265,A -85,B 0,C 180,E1 -16190.849,E2 -16190.849} C_VEL
LIN {X 0,Y 298.706,Z 190.276,A -85,B 0,C 180,E1 -16191.229,E2 -16191.229} C_VEL
LIN {X 0,Y 298.637,Z 190.283,A -85,B 0,C 180,E1 -16194.598,E2 -16194.598} C_VEL
LIN {X 0,Y 298.924,Z 190.248,A -85,B 0,C 180,E1 -16198.653,E2 -16198.653} C_VEL
LIN {X 0,Y 298.924,Z 190.251,A -85,B 0,C 180,E1 -16201.347,E2 -16201.347} C_VEL
LIN {X 0,Y 298.638,Z 190.285,A -85,B 0,C 180,E1 -16205.401,E2 -16205.401} C_VEL
LIN {X 0,Y 298.708,Z 190.28,A -85,B 0,C 180,E1 -16208.82,E2 -16208.82} C_VEL
LIN {X 0,Y 298.556,Z 190.296,A -85,B 0,C 180,E1 -16212.231,E2 -16212.231} C_VEL
LIN {X 0,Y 298.607,Z 190.289,A -85,B 0,C 180,E1 -16215.209,E2 -16215.209} C_VEL
LIN {X 0,Y 298.527,Z 190.298,A -85,B 0,C 180,E1 -16219.244,E2 -16219.244} C_VEL
LIN {X 0,Y 298.43,Z 190.31,A -85,B 0,C 180,E1 -16223.6,E2 -16223.6} C_VEL
LIN {X 0,Y 298.49,Z 190.304,A -85,B 0,C 180,E1 -16226.574,E2 -16226.574} C_VEL
LIN {X 0,Y 298.418,Z 190.314,A -85,B 0,C 180,E1 -16229.641,E2 -16229.641} C_VEL
LIN {X 0,Y 298.396,Z 190.316,A -85,B 0,C 180,E1 -16232.8,E2 -16232.8} C_VEL
LIN {X 0,Y 298.429,Z 190.312,A -85,B 0,C 180,E1 -16236.803,E2 -16236.803} C_VEL
LIN {X 0,Y 298.388,Z 190.319,A -85,B 0,C 180,E1 -16241.088,E2 -16241.088} C_VEL
LIN {X 0,Y 298.432,Z 190.376,A -85,B 0,C 180,E1 -16242.844,E2 -16242.844} C_VEL
LIN {X 0,Y 299.226,Z 195,A -85,B 0,C 180,E1 -16247.068,E2 -16247.068} C_VEL
LIN {X 0,Y 299.928,Z 199.347,A -85,B 0,C 180,E1 -16250.752,E2 -16250.752} C_VEL
LIN {X 0,Y 300.197,Z 203.698,A -85,B 0,C 180,E1 -16254.177,E2 -16254.177} C_VEL
LIN {X 0,Y 299.629,Z 208.327,A -85,B 0,C 180,E1 -16257.608,E2 -16257.608} C_VEL
LIN {X 0,Y 298.94,Z 213.33,A -85,B 0,C 180,E1 -16261.187,E2 -16261.187} C_VEL
LIN {X 0,Y 298.175,Z 219.33,A -85,B 0,C 180,E1 -16265.42,E2 -16265.42} C_VEL
LIN {X 0,Y 301.399,Z 232.883,A -85,B 0,C 180,E1 -16266.301,E2 -16266.301} C_VEL
LIN {X 0,Y 303.518,Z 245.176,A -85,B 0,C 180,E1 -16267.298,E2 -16267.298} C_VEL
LIN {X 0,Y 304.821,Z 255.953,A -85,B 0,C 180,E1 -16268.352,E2 -16268.352} C_VEL
LIN {X 0,Y 305.401,Z 264.155,A -85,B 0,C 180,E1 -16269.279,E2 -16269.279} C_VEL
LIN {X 0,Y 303.885,Z 274.771,A -85,B 0,C 180,E1 -16270.582,E2 -16270.582} C_VEL
LIN {X 0,Y 302.379,Z 284.475,A -85,B 0,C 180,E1 -16272.063,E2 -16272.063} C_VEL
LIN {X 0,Y 301.01,Z 293.321,A -85,B 0,C 180,E1 -16273.729,E2 -16273.729} C_VEL
LIN {X 0,Y 299.793,Z 300.626,A -85,B 0,C 180,E1 -16275.403,E2 -16275.403} C_VEL
LIN {X 0,Y 298.537,Z 307.819,A -85,B 0,C 180,E1 -16277.422,E2 -16277.422} C_VEL
LIN {X 0,Y 297.8,Z 312.679,A -85,B 0,C 180,E1 -16279.117,E2 -16279.117} C_VEL
LIN {X 0,Y 297.161,Z 317.404,A -85,B 0,C 180,E1 -16281.157,E2 -16281.157} C_VEL
LIN {X 0,Y 296.755,Z 321.017,A -85,B 0,C 180,E1 -16283.199,E2 -16283.199} C_VEL
LIN {X 0,Y 296.601,Z 322.881,A -85,B 0,C 180,E1 -16284.561,E2 -16284.561} C_VEL
LIN {X 0,Y 296.546,Z 324.28,A -85,B 0,C 180,E1 -16285.923,E2 -16285.923} C_VEL
LIN {X 0,Y 296.536,Z 325.28,A -85,B 0,C 180,E1 -16287.283,E2 -16287.283} C_VEL
LIN {X 0,Y 296.48,Z 325.888,A -85,B 0,C 180,E1 -16288.641,E2 -16288.641} C_VEL
LIN {X 0,Y 296.487,Z 326.104,A -85,B 0,C 180,E1 -16290,E2 -16290} C_VEL
LIN {X 0,Y 296.48,Z 325.884,A -85,B 0,C 180,E1 -16291.358,E2 -16291.358} C_VEL
LIN {X 0,Y 296.535,Z 325.274,A -85,B 0,C 180,E1 -16292.717,E2 -16292.717} C_VEL
LIN {X 0,Y 296.547,Z 324.273,A -85,B 0,C 180,E1 -16294.077,E2 -16294.077} C_VEL
LIN {X 0,Y 296.623,Z 322.582,A -85,B 0,C 180,E1 -16295.66,E2 -16295.66} C_VEL
LIN {X 0,Y 296.981,Z 318.692,A -85,B 0,C 180,E1 -16298.163,E2 -16298.163} C_VEL
LIN {X 0,Y 297.546,Z 314.342,A -85,B 0,C 180,E1 -16300.203,E2 -16300.203} C_VEL
LIN {X 0,Y 298.338,Z 308.802,A -85,B 0,C 180,E1 -16302.24,E2 -16302.24} C_VEL
LIN {X 0,Y 299.542,Z 301.895,A -85,B 0,C 180,E1 -16304.262,E2 -16304.262} C_VEL
LIN {X 0,Y 301.016,Z 293.253,A -85,B 0,C 180,E1 -16306.27,E2 -16306.27} C_VEL
LIN {X 0,Y 302.384,Z 284.391,A -85,B 0,C 180,E1 -16307.936,E2 -16307.936} C_VEL
LIN {X 0,Y 303.868,Z 274.668,A -85,B 0,C 180,E1 -16309.418,E2 -16309.418} C_VEL
LIN {X 0,Y 305.313,Z 264.029,A -85,B 0,C 180,E1 -16310.727,E2 -16310.727} C_VEL
LIN {X 0,Y 304.436,Z 252.206,A -85,B 0,C 180,E1 -16312.02,E2 -16312.02} C_VEL
LIN {X 0,Y 302.697,Z 239.758,A -85,B 0,C 180,E1 -16313.145,E2 -16313.145} C_VEL
LIN {X 0,Y 299.998,Z 226.852,A -85,B 0,C 180,E1 -16314.105,E2 -16314.105} C_VEL
LIN {X 0,Y 298.173,Z 219.324,A -85,B 0,C 180,E1 -16314.566,E2 -16314.566} C_VEL
LIN {X 0,Y 298.938,Z 213.305,A -85,B 0,C 180,E1 -16318.813,E2 -16318.813} C_VEL
LIN {X 0,Y 299.671,Z 207.966,A -85,B 0,C 180,E1 -16322.643,E2 -16322.643} C_VEL
LIN {X 0,Y 300.211,Z 203.669,A -85,B 0,C 180,E1 -16325.82,E2 -16325.82} C_VEL
LIN {X 0,Y 299.934,Z 199.192,A -85,B 0,C 180,E1 -16329.353,E2 -16329.353} C_VEL
LIN {X 0,Y 299.163,Z 194.598,A -85,B 0,C 180,E1 -16333.259,E2 -16333.259} C_VEL
LIN {X 0,Y 298.44,Z 190.315,A -85,B 0,C 180,E1 -16337.273,E2 -16337.273} C_VEL
LIN {X 0,Y 298.394,Z 190.317,A -85,B 0,C 180,E1 -16341.008,E2 -16341.008} C_VEL
LIN {X 0,Y 298.404,Z 190.316,A -85,B 0,C 180,E1 -16343.928,E2 -16343.928} C_VEL
LIN {X 0,Y 298.393,Z 190.315,A -85,B 0,C 180,E1 -16347.199,E2 -16347.199} C_VEL
LIN {X 0,Y 298.425,Z 190.311,A -85,B 0,C 180,E1 -16350.616,E2 -16350.616} C_VEL
LIN {X 0,Y 298.481,Z 190.305,A -85,B 0,C 180,E1 -16353.474,E2 -16353.474} C_VEL
LIN {X 0,Y 298.429,Z 190.311,A -85,B 0,C 180,E1 -16356.699,E2 -16356.699} C_VEL
LIN {X 0,Y 298.537,Z 190.297,A -85,B 0,C 180,E1 -16360.757,E2 -16360.757} C_VEL
LIN {X 0,Y 298.592,Z 190.291,A -85,B 0,C 180,E1 -16364.995,E2 -16364.995} C_VEL
LIN {X 0,Y 298.581,Z 190.291,A -85,B 0,C 180,E1 -16369.146,E2 -16369.146} C_VEL
LIN {X 0,Y 298.695,Z 190.276,A -85,B 0,C 180,E1 -16371.884,E2 -16371.884} C_VEL
LIN {X 0,Y 298.635,Z 190.285,A -85,B 0,C 180,E1 -16374.599,E2 -16374.599} C_VEL
LIN {X 0,Y 298.921,Z 190.25,A -85,B 0,C 180,E1 -16378.653,E2 -16378.653} C_VEL
LIN {X 0,Y 298.921,Z 190.249,A -85,B 0,C 180,E1 -16381.347,E2 -16381.347} C_VEL
LIN {X 0,Y 298.635,Z 190.284,A -85,B 0,C 180,E1 -16385.402,E2 -16385.402} C_VEL
LIN {X 0,Y 298.705,Z 190.277,A -85,B 0,C 180,E1 -16388.82,E2 -16388.82} C_VEL
LIN {X 0,Y 298.55,Z 190.294,A -85,B 0,C 180,E1 -16393.616,E2 -16393.616} C_VEL
LIN {X 0,Y 298.547,Z 190.298,A -85,B 0,C 180,E1 -16396.409,E2 -16396.409} C_VEL
LIN {X 0,Y 298.51,Z 190.301,A -85,B 0,C 180,E1 -16399.655,E2 -16399.655} C_VEL
LIN {X 0,Y 298.456,Z 190.309,A -85,B 0,C 180,E1 -16403.598,E2 -16403.598} C_VEL
LIN {X 0,Y 298.485,Z 190.303,A -85,B 0,C 180,E1 -16406.575,E2 -16406.575} C_VEL
LIN {X 0,Y 298.419,Z 190.314,A -85,B 0,C 180,E1 -16409.641,E2 -16409.641} C_VEL
LIN {X 0,Y 298.394,Z 190.314,A -85,B 0,C 180,E1 -16412.801,E2 -16412.801} C_VEL
LIN {X 0,Y 298.427,Z 190.311,A -85,B 0,C 180,E1 -16416.803,E2 -16416.803} C_VEL
LIN {X 0,Y 298.386,Z 190.32,A -85,B 0,C 180,E1 -16421.088,E2 -16421.088} C_VEL
LIN {X 0,Y 298.398,Z 190.319,A -85,B 0,C 180,E1 -16423.104,E2 -16423.104} C_VEL
LIN {X 0,Y 298.402,Z 190.317,A -85,B 0,C 180,E1 -16426.921,E2 -16426.921} C_VEL
LIN {X 0,Y 298.395,Z 190.318,A -85,B 0,C 180,E1 -16431.009,E2 -16431.009} C_VEL
LIN {X 0,Y 298.513,Z 192.636,A -85,B 0,C 180,E1 -16433.944,E2 -16433.944} C_VEL
LIN {X 0,Y 298.364,Z 195.657,A -85,B 0,C 180,E1 -16437.197,E2 -16437.197} C_VEL
LIN {X 0,Y 298.129,Z 199.077,A -85,B 0,C 180,E1 -16440.719,E2 -16440.719} C_VEL
LIN {X 0,Y 297.745,Z 203.333,A -85,B 0,C 180,E1 -16444.858,E2 -16444.858} C_VEL
LIN {X 0,Y 297.739,Z 203.972,A -85,B 0,C 180,E1 -16445.469,E2 -16445.469} C_VEL
LIN {X 0,Y 301.956,Z 218.196,A -85,B 0,C 180,E1 -16446.529,E2 -16446.529} C_VEL
LIN {X 0,Y 304.787,Z 230.712,A -85,B 0,C 180,E1 -16447.654,E2 -16447.654} C_VEL
LIN {X 0,Y 306.573,Z 241.731,A -85,B 0,C 180,E1 -16448.835,E2 -16448.835} C_VEL
LIN {X 0,Y 305.467,Z 252.075,A -85,B 0,C 180,E1 -16449.987,E2 -16449.987} C_VEL
LIN {X 0,Y 303.98,Z 262.518,A -85,B 0,C 180,E1 -16451.427,E2 -16451.427} C_VEL
LIN {X 0,Y 302.539,Z 272.341,A -85,B 0,C 180,E1 -16453.12,E2 -16453.12} C_VEL
LIN {X 0,Y 301.167,Z 280.204,A -85,B 0,C 180,E1 -16454.78,E2 -16454.78} C_VEL
LIN {X 0,Y 299.781,Z 287.886,A -85,B 0,C 180,E1 -16456.787,E2 -16456.787} C_VEL
LIN {X 0,Y 298.483,Z 294.938,A -85,B 0,C 180,E1 -16459.143,E2 -16459.143} C_VEL
